gfCNCPoint6[1225] = {X 338.7767, Y 49.3353, Z -8.0000, A 0.000, B 0.000, C 0.000 }
gfCNCPoint6[1226] = {X 336.8016, Y 48.5824, Z -8.0000, A 0.000, B 0.000, C 0.000 }
gfCNCPoint6[1227] = {X 334.8992, Y 47.6612, Z -8.0000, A 0.000, B 0.000, C 0.000 }
gfCNCPoint6[1228] = {X 333.3419, Y 46.7043, Z -8.0000, A 0.000, B 0.000, C 0.000 }
gfCNCPoint6[1229] = {X 331.8606, Y 45.6336, Z -8.0000, A 0.000, B 0.000, C 0.000 }
gfCNCPoint6[1230] = {X 330.4636, Y 44.4550, Z -8.0000, A 0.000, B 0.000, C 0.000 }
gfCNCPoint6[1231] = {X 329.4664, Y 44.4078, Z -8.0000, A 0.000, B 0.000, C 0.000 }
gfCNCPoint6[1232] = {X 328.4996, Y 44.1587, Z -8.0000, A 0.000, B 0.000, C 0.000 }
gfCNCPoint6[1233] = {X 327.6038, Y 43.7181, Z -8.0000, A 0.000, B 0.000, C 0.000 }
gfCNCPoint6[1234] = {X 326.8164, Y 43.1044, Z -8.0000, A 0.000, B 0.000, C 0.000 }
gfCNCPoint6[1235] = {X 326.1897, Y 42.4934, Z -8.0000, A 0.000, B 0.000, C 0.000 }
gfCNCPoint6[1236] = {X 325.5686, Y 41.7541, Z -8.0000, A 0.000, B 0.000, C 0.000 }
gfCNCPoint6[1237] = {X 325.1052, Y 40.9070, Z -8.0000, A 0.000, B 0.000, C 0.000 }
gfCNCPoint6[1238] = {X 324.8177, Y 39.9852, Z -8.0000, A 0.000, B 0.000, C 0.000 }
gfCNCPoint6[1239] = {X 324.7172, Y 39.0249, Z -8.0000, A 0.000, B 0.000, C 0.000 }
gfCNCPoint6[1240] = {X 324.8079, Y 38.0635, Z -8.0000, A 0.000, B 0.000, C 0.000 }
gfCNCPoint6[1241] = {X 325.0860, Y 37.1389, Z -8.0000, A 0.000, B 0.000, C 0.000 }
gfCNCPoint6[1242] = {X 325.5408, Y 36.2871, Z -8.0000, A 0.000, B 0.000, C 0.000 }
gfCNCPoint6[1243] = {X 329.7765, Y 29.9537, Z -8.0000, A 0.000, B 0.000, C 0.000 }
gfCNCPoint6[1244] = {X 330.4614, Y 29.1399, Z -8.0000, A 0.000, B 0.000, C 0.000 }
gfCNCPoint6[1245] = {X 331.3063, Y 28.4938, Z -8.0000, A 0.000, B 0.000, C 0.000 }
gfCNCPoint6[1246] = {X 332.2712, Y 28.0462, Z -8.0000, A 0.000, B 0.000, C 0.000 }
gfCNCPoint6[1247] = {X 333.3101, Y 27.8182, Z -8.0000, A 0.000, B 0.000, C 0.000 }
gfCNCPoint6[1248] = {X 334.3737, Y 27.8207, Z -8.0000, A 0.000, B 0.000, C 0.000 }
gfCNCPoint6[1249] = {X 335.4115, Y 28.0536, Z -8.0000, A 0.000, B 0.000, C 0.000 }
gfCNCPoint6[1250] = {X 336.3742, Y 28.5058, Z -8.0000, A 0.000, B 0.000, C 0.000 }
gfCNCPoint6[1251] = {X 337.2161, Y 29.1558, Z -8.0000, A 0.000, B 0.000, C 0.000 }
gfCNCPoint6[1252] = {X 337.8208, Y 29.7387, Z -8.0000, A 0.000, B 0.000, C 0.000 }
gfCNCPoint6[1253] = {X 338.4966, Y 30.5667, Z -8.0000, A 0.000, B 0.000, C 0.000 }
gfCNCPoint6[1254] = {X 338.9759, Y 31.5219, Z -8.0000, A 0.000, B 0.000, C 0.000 }
gfCNCPoint6[1255] = {X 339.2358, Y 32.5585, Z -8.0000, A 0.000, B 0.000, C 0.000 }
gfCNCPoint6[1256] = {X 339.2638, Y 33.6268, Z -8.0000, A 0.000, B 0.000, C 0.000 }
gfCNCPoint6[1257] = {X 339.8716, Y 34.1825, Z -8.0000, A 0.000, B 0.000, C 0.000 }
gfCNCPoint6[1258] = {X 340.9509, Y 35.0427, Z -8.0000, A 0.000, B 0.000, C 0.000 }
gfCNCPoint6[1259] = {X 342.1372, Y 35.7481, Z -8.0000, A 0.000, B 0.000, C 0.000 }
gfCNCPoint6[1260] = {X 343.4085, Y 36.2856, Z -8.0000, A 0.000, B 0.000, C 0.000 }
gfCNCPoint6[1261] = {X 344.7410, Y 36.6452, Z -8.0000, A 0.000, B 0.000, C 0.000 }
gfCNCPoint6[1262] = {X 346.1100, Y 36.8203, Z -8.0000, A 0.000, B 0.000, C 0.000 }
gfCNCPoint6[1263] = {X 347.4901, Y 36.8075, Z -8.0000, A 0.000, B 0.000, C 0.000 }
gfCNCPoint6[1264] = {X 348.8397, Y 36.6262, Z -8.0000, A 0.000, B 0.000, C 0.000 }
gfCNCPoint6[1265] = {X 350.1418, Y 36.2276, Z -8.0000, A 0.000, B 0.000, C 0.000 }
gfCNCPoint6[1266] = {X 351.3616, Y 35.6223, Z -8.0000, A 0.000, B 0.000, C 0.000 }
gfCNCPoint6[1267] = {X 352.4665, Y 34.8263, Z -8.0000, A 0.000, B 0.000, C 0.000 }
gfCNCPoint6[1268] = {X 353.5670, Y 33.7568, Z -8.0000, A 0.000, B 0.000, C 0.000 }
gfCNCPoint6[1269] = {X 354.5194, Y 32.5535, Z -8.0000, A 0.000, B 0.000, C 0.000 }
gfCNCPoint6[1270] = {X 355.3077, Y 31.2368, Z -8.0000, A 0.000, B 0.000, C 0.000 }
gfCNCPoint6[1271] = {X 355.9184, Y 29.8290, Z -8.0000, A 0.000, B 0.000, C 0.000 }
gfCNCPoint6[1272] = {X 356.3412, Y 28.3538, Z -8.0000, A 0.000, B 0.000, C 0.000 }
gfCNCPoint6[1273] = {X 356.6058, Y 26.7186, Z -8.0000, A 0.000, B 0.000, C 0.000 }
gfCNCPoint6[1274] = {X 356.7135, Y 25.0657, Z -8.0000, A 0.000, B 0.000, C 0.000 }
gfCNCPoint6[1275] = {X 356.6634, Y 23.4100, Z -8.0000, A 0.000, B 0.000, C 0.000 }
gfCNCPoint6[1276] = {X 356.4559, Y 21.7666, Z -8.0000, A 0.000, B 0.000, C 0.000 }
gfCNCPoint6[1277] = {X 356.1193, Y 20.3212, Z -8.0000, A 0.000, B 0.000, C 0.000 }
gfCNCPoint6[1278] = {X 355.5958, Y 18.9324, Z -8.0000, A 0.000, B 0.000, C 0.000 }
gfCNCPoint6[1279] = {X 354.8945, Y 17.6245, Z -8.0000, A 0.000, B 0.000, C 0.000 }
gfCNCPoint6[1280] = {X 354.0274, Y 16.4200, Z -8.0000, A 0.000, B 0.000, C 0.000 }
gfCNCPoint6[1281] = {X 353.2099, Y 15.5491, Z -8.0000, A 0.000, B 0.000, C 0.000 }
gfCNCPoint6[1282] = {X 352.2795, Y 14.8000, Z -8.0000, A 0.000, B 0.000, C 0.000 }
gfCNCPoint6[1283] = {X 351.2542, Y 14.1872, Z -8.0000, A 0.000, B 0.000, C 0.000 }
gfCNCPoint6[1284] = {X 350.1538, Y 13.7227, Z -8.0000, A 0.000, B 0.000, C 0.000 }
gfCNCPoint6[1285] = {X 348.9996, Y 13.4152, Z -8.0000, A 0.000, B 0.000, C 0.000 }
gfCNCPoint6[1286] = {X 347.3622, Y 13.2074, Z -8.0000, A 0.000, B 0.000, C 0.000 }
gfCNCPoint6[1287] = {X 345.7117, Y 13.2121, Z -8.0000, A 0.000, B 0.000, C 0.000 }
gfCNCPoint6[1288] = {X 344.0755, Y 13.4290, Z -8.0000, A 0.000, B 0.000, C 0.000 }
gfCNCPoint6[1289] = {X 342.4808, Y 13.8547, Z -8.0000, A 0.000, B 0.000, C 0.000 }
gfCNCPoint6[1290] = {X 340.9542, Y 14.4820, Z -8.0000, A 0.000, B 0.000, C 0.000 }
gfCNCPoint6[1291] = {X 339.5209, Y 15.3006, Z -8.0000, A 0.000, B 0.000, C 0.000 }
gfCNCPoint6[1292] = {X 339.4270, Y 16.1861, Z -8.0000, A 0.000, B 0.000, C 0.000 }
gfCNCPoint6[1293] = {X 339.1738, Y 17.0397, Z -8.0000, A 0.000, B 0.000, C 0.000 }
gfCNCPoint6[1294] = {X 338.7696, Y 17.8332, Z -8.0000, A 0.000, B 0.000, C 0.000 }
gfCNCPoint6[1295] = {X 338.2280, Y 18.5400, Z -8.0000, A 0.000, B 0.000, C 0.000 }
gfCNCPoint6[1296] = {X 337.5670, Y 19.1366, Z -8.0000, A 0.000, B 0.000, C 0.000 }
gfCNCPoint6[1297] = {X 336.8400, Y 19.6716, Z -8.0000, A 0.000, B 0.000, C 0.000 }
gfCNCPoint6[1298] = {X 335.9171, Y 20.1909, Z -8.0000, A 0.000, B 0.000, C 0.000 }
gfCNCPoint6[1299] = {X 334.9039, Y 20.4988, Z -8.0000, A 0.000, B 0.000, C 0.000 }
gfCNCPoint6[1300] = {X 333.8481, Y 20.5809, Z -8.0000, A 0.000, B 0.000, C 0.000 }
gfCNCPoint6[1301] = {X 332.7995, Y 20.4334, Z -8.0000, A 0.000, B 0.000, C 0.000 }
gfCNCPoint6[1302] = {X 331.8074, Y 20.0631, Z -8.0000, A 0.000, B 0.000, C 0.000 }
gfCNCPoint6[1303] = {X 330.9186, Y 19.4876, Z -8.0000, A 0.000, B 0.000, C 0.000 }
gfCNCPoint6[1304] = {X 330.1748, Y 18.7338, Z -8.0000, A 0.000, B 0.000, C 0.000 }
gfCNCPoint6[1305] = {X 329.6111, Y 17.8373, Z -8.0000, A 0.000, B 0.000, C 0.000 }
gfCNCPoint6[1306] = {X 326.0906, Y 10.5950, Z -8.0000, A 0.000, B 0.000, C 0.000 }
gfCNCPoint6[1307] = {X 325.7555, Y 9.6856, Z -8.0000, A 0.000, B 0.000, C 0.000 }
gfCNCPoint6[1308] = {X 325.6067, Y 8.7279, Z -8.0000, A 0.000, B 0.000, C 0.000 }
gfCNCPoint6[1309] = {X 325.6502, Y 7.7596, Z -8.0000, A 0.000, B 0.000, C 0.000 }
gfCNCPoint6[1310] = {X 325.8842, Y 6.8191, Z -8.0000, A 0.000, B 0.000, C 0.000 }
gfCNCPoint6[1311] = {X 326.2994, Y 5.9433, Z -8.0000, A 0.000, B 0.000, C 0.000 }
gfCNCPoint6[1312] = {X 326.9295, Y 5.1131, Z -8.0000, A 0.000, B 0.000, C 0.000 }
gfCNCPoint6[1313] = {X 327.7216, Y 4.4356, Z -8.0000, A 0.000, B 0.000, C 0.000 }
gfCNCPoint6[1314] = {X 328.3968, Y 3.9733, Z -8.0000, A 0.000, B 0.000, C 0.000 }
gfCNCPoint6[1315] = {X 329.3289, Y 3.4830, Z -8.0000, A 0.000, B 0.000, C 0.000 }
gfCNCPoint6[1316] = {X 330.3446, Y 3.2042, Z -8.0000, A 0.000, B 0.000, C 0.000 }
gfCNCPoint6[1317] = {X 331.3964, Y 3.1497, Z -8.0000, A 0.000, B 0.000, C 0.000 }
gfCNCPoint6[1318] = {X 332.4354, Y 3.3223, Z -8.0000, A 0.000, B 0.000, C 0.000 }
gfCNCPoint6[1319] = {X 333.3715, Y 2.7957, Z -8.0000, A 0.000, B 0.000, C 0.000 }
gfCNCPoint6[1320] = {X 334.3268, Y 2.3048, Z -8.0000, A 0.000, B 0.000, C 0.000 }
gfCNCPoint6[1321] = {X 334.5381, Y 2.7358, Z -8.0000, A 0.000, B 0.000, C 0.000 }
gfCNCPoint6[1322] = {X 335.0034, Y 2.5130, Z -8.0000, A 0.000, B 0.000, C 0.000 }
gfCNCPoint6[1323] = {X 335.4728, Y 2.2988, Z -8.0000, A 0.000, B 0.000, C 0.000 }
gfCNCPoint6[1324] = {X 335.8480, Y 2.1318, Z -8.0000, A 0.000, B 0.000, C 0.000 }
gfCNCPoint6[1325] = {X 337.9512, Y 1.3113, Z -8.0000, A 0.000, B 0.000, C 0.000 }
gfCNCPoint6[1326] = {X 340.1169, Y 0.6737, Z -8.0000, A 0.000, B 0.000, C 0.000 }
gfCNCPoint6[1327] = {X 342.3292, Y 0.2238, Z -8.0000, A 0.000, B 0.000, C 0.000 }
gfCNCPoint6[1328] = {X 344.5719, Y -0.0351, Z -8.0000, A 0.000, B 0.000, C 0.000 }
gfCNCPoint6[1329] = {X 346.8285, Y -0.1013, Z -8.0000, A 0.000, B 0.000, C 0.000 }
gfCNCPoint6[1330] = {X 349.0825, Y 0.0259, Z -8.0000, A 0.000, B 0.000, C 0.000 }
gfCNCPoint6[1331] = {X 351.3173, Y 0.3455, Z -8.0000, A 0.000, B 0.000, C 0.000 }
gfCNCPoint6[1332] = {X 351.8894, Y 0.4533, Z -8.0000, A 0.000, B 0.000, C 0.000 }
gfCNCPoint6[1333] = {X 354.0191, Y 0.9988, Z -8.0000, A 0.000, B 0.000, C 0.000 }
gfCNCPoint6[1334] = {X 356.0806, Y 1.7630, Z -8.0000, A 0.000, B 0.000, C 0.000 }
gfCNCPoint6[1335] = {X 358.0513, Y 2.7375, Z -8.0000, A 0.000, B 0.000, C 0.000 }
gfCNCPoint6[1336] = {X 359.9100, Y 3.9117, Z -8.0000, A 0.000, B 0.000, C 0.000 }
gfCNCPoint6[1337] = {X 361.6364, Y 5.2730, Z -8.0000, A 0.000, B 0.000, C 0.000 }
gfCNCPoint6[1338] = {X 363.2118, Y 6.8065, Z -8.0000, A 0.000, B 0.000, C 0.000 }
gfCNCPoint6[1339] = {X 364.7640, Y 8.6820, Z -8.0000, A 0.000, B 0.000, C 0.000 }
gfCNCPoint6[1340] = {X 366.1253, Y 10.7002, Z -8.0000, A 0.000, B 0.000, C 0.000 }
gfCNCPoint6[1341] = {X 367.2828, Y 12.8419, Z -8.0000, A 0.000, B 0.000, C 0.000 }
gfCNCPoint6[1342] = {X 368.2254, Y 15.0864, Z -8.0000, A 0.000, B 0.000, C 0.000 }
gfCNCPoint6[1343] = {X 368.9440, Y 17.4124, Z -8.0000, A 0.000, B 0.000, C 0.000 }
gfCNCPoint6[1344] = {X 369.4273, Y 19.7106, Z -8.0000, A 0.000, B 0.000, C 0.000 }
gfCNCPoint6[1345] = {X 369.7390, Y 22.0383, Z -8.0000, A 0.000, B 0.000, C 0.000 }
gfCNCPoint6[1346] = {X 369.8772, Y 24.3826, Z -8.0000, A 0.000, B 0.000, C 0.000 }
gfCNCPoint6[1347] = {X 369.8413, Y 26.7308, Z -8.0000, A 0.000, B 0.000, C 0.000 }
gfCNCPoint6[1348] = {X 369.6314, Y 29.0699, Z -8.0000, A 0.000, B 0.000, C 0.000 }
gfCNCPoint6[1349] = {X 369.2488, Y 31.3870, Z -8.0000, A 0.000, B 0.000, C 0.000 }
gfCNCPoint6[1350] = {X 368.7229, Y 33.4980, Z -8.0000, A 0.000, B 0.000, C 0.000 }
gfCNCPoint6[1351] = {X 368.0128, Y 35.5544, Z -8.0000, A 0.000, B 0.000, C 0.000 }
gfCNCPoint6[1352] = {X 367.1239, Y 37.5400, Z -8.0000, A 0.000, B 0.000, C 0.000 }
gfCNCPoint6[1353] = {X 366.0631, Y 39.4394, Z -8.0000, A 0.000, B 0.000, C 0.000 }
gfCNCPoint6[1354] = {X 364.8388, Y 41.2378, Z -8.0000, A 0.000, B 0.000, C 0.000 }
gfCNCPoint6[1355] = {X 364.7204, Y 41.3994, Z -8.0000, A 0.000, B 0.000, C 0.000 }
gfCNCPoint6[1356] = {X 363.4201, Y 42.9682, Z -8.0000, A 0.000, B 0.000, C 0.000 }
gfCNCPoint6[1357] = {X 361.9805, Y 44.4103, Z -8.0000, A 0.000, B 0.000, C 0.000 }
gfCNCPoint6[1358] = {X 360.4141, Y 45.7135, Z -8.0000, A 0.000, B 0.000, C 0.000 }
gfCNCPoint6[1359] = {X 358.7341, Y 46.8667, Z -8.0000, A 0.000, B 0.000, C 0.000 }
gfCNCPoint6[1360] = {X 356.9549, Y 47.8599, Z -8.0000, A 0.000, B 0.000, C 0.000 }
gfCNCPoint6[1361] = {X 356.2499, Y 48.1934, Z -8.0000, A 0.000, B 0.000, C 0.000 }
gfCNCPoint6[1362] = {X 354.0456, Y 49.0158, Z -8.0000, A 0.000, B 0.000, C 0.000 }
gfCNCPoint6[1363] = {X 351.7691, Y 49.6098, Z -8.0000, A 0.000, B 0.000, C 0.000 }
gfCNCPoint6[1364] = {X 349.4439, Y 49.9692, Z -8.0000, A 0.000, B 0.000, C 0.000 }
gfCNCPoint6[1365] = {X 347.0943, Y 50.0903, Z -8.0000, A 0.000, B 0.000, C 0.000 }
gfCNCPoint6[1366] = {X 345.0202, Y 50.0551, Z -8.0000, A 0.000, B 0.000, C 0.000 }
gfCNCPoint6[1367] = {X 342.9569, Y 49.8401, Z -8.0000, A 0.000, B 0.000, C 0.000 }
gfCNCPoint6[1368] = {X 340.9201, Y 49.4470, Z -8.0000, A 0.000, B 0.000, C 0.000 }
gfCNCPoint6[1369] = {X 338.9250, Y 48.8787, Z -8.0000, A 0.000, B 0.000, C 0.000 }
gfCNCPoint6[1370] = {X 336.9867, Y 48.1394, Z -8.0000, A 0.000, B 0.000, C 0.000 }
gfCNCPoint6[1371] = {X 335.1199, Y 47.2348, Z -8.0000, A 0.000, B 0.000, C 0.000 }
gfCNCPoint6[1372] = {X 333.5416, Y 46.2605, Z -8.0000, A 0.000, B 0.000, C 0.000 }
gfCNCPoint6[1373] = {X 332.0435, Y 45.1668, Z -8.0000, A 0.000, B 0.000, C 0.000 }
gfCNCPoint6[1374] = {X 330.6346, Y 43.9603, Z -8.0000, A 0.000, B 0.000, C 0.000 }
gfCNCPoint6[1375] = {X 329.6760, Y 43.9518, Z -8.0000, A 0.000, B 0.000, C 0.000 }
gfCNCPoint6[1376] = {X 328.7421, Y 43.7359, Z -8.0000, A 0.000, B 0.000, C 0.000 }
gfCNCPoint6[1377] = {X 327.8770, Y 43.3228, Z -8.0000, A 0.000, B 0.000, C 0.000 }
gfCNCPoint6[1378] = {X 327.1220, Y 42.7322, Z -8.0000, A 0.000, B 0.000, C 0.000 }
gfCNCPoint6[1379] = {X 326.5249, Y 42.1498, Z -8.0000, A 0.000, B 0.000, C 0.000 }
gfCNCPoint6[1380] = {X 325.8848, Y 41.3619, Z -8.0000, A 0.000, B 0.000, C 0.000 }
gfCNCPoint6[1381] = {X 325.4424, Y 40.4483, Z -8.0000, A 0.000, B 0.000, C 0.000 }
gfCNCPoint6[1382] = {X 325.2210, Y 39.4576, Z -8.0000, A 0.000, B 0.000, C 0.000 }
gfCNCPoint6[1383] = {X 325.2326, Y 38.4426, Z -8.0000, A 0.000, B 0.000, C 0.000 }
gfCNCPoint6[1384] = {X 325.4765, Y 37.4572, Z -8.0000, A 0.000, B 0.000, C 0.000 }
gfCNCPoint6[1385] = {X 325.9397, Y 36.5539, Z -8.0000, A 0.000, B 0.000, C 0.000 }
gfCNCPoint6[1386] = {X 330.1988, Y 30.1861, Z -8.0000, A 0.000, B 0.000, C 0.000 }
gfCNCPoint6[1387] = {X 330.8195, Y 29.4619, Z -8.0000, A 0.000, B 0.000, C 0.000 }
gfCNCPoint6[1388] = {X 331.5816, Y 28.8884, Z -8.0000, A 0.000, B 0.000, C 0.000 }
gfCNCPoint6[1389] = {X 332.4494, Y 28.4927, Z -8.0000, A 0.000, B 0.000, C 0.000 }
gfCNCPoint6[1390] = {X 333.3822, Y 28.2932, Z -8.0000, A 0.000, B 0.000, C 0.000 }
gfCNCPoint6[1391] = {X 334.3359, Y 28.2995, Z -8.0000, A 0.000, B 0.000, C 0.000 }
gfCNCPoint6[1392] = {X 335.2659, Y 28.5111, Z -8.0000, A 0.000, B 0.000, C 0.000 }
gfCNCPoint6[1393] = {X 336.1285, Y 28.9182, Z -8.0000, A 0.000, B 0.000, C 0.000 }
gfCNCPoint6[1394] = {X 336.8831, Y 29.5015, Z -8.0000, A 0.000, B 0.000, C 0.000 }
gfCNCPoint6[1395] = {X 337.4845, Y 30.0811, Z -8.0000, A 0.000, B 0.000, C 0.000 }
gfCNCPoint6[1396] = {X 338.1249, Y 30.8764, Z -8.0000, A 0.000, B 0.000, C 0.000 }
gfCNCPoint6[1397] = {X 338.5647, Y 31.7978, Z -8.0000, A 0.000, B 0.000, C 0.000 }
gfCNCPoint6[1398] = {X 338.7803, Y 32.7959, Z -8.0000, A 0.000, B 0.000, C 0.000 }
gfCNCPoint6[1399] = {X 338.7601, Y 33.8167, Z -8.0000, A 0.000, B 0.000, C 0.000 }
gfCNCPoint6[1400] = {X 339.5477, Y 34.5368, Z -8.0000, A 0.000, B 0.000, C 0.000 }
gfCNCPoint6[1401] = {X 340.6406, Y 35.4108, Z -8.0000, A 0.000, B 0.000, C 0.000 }
gfCNCPoint6[1402] = {X 341.8390, Y 36.1333, Z -8.0000, A 0.000, B 0.000, C 0.000 }
gfCNCPoint6[1403] = {X 343.1221, Y 36.6917, Z -8.0000, A 0.000, B 0.000, C 0.000 }
gfCNCPoint6[1404] = {X 344.4675, Y 37.0763, Z -8.0000, A 0.000, B 0.000, C 0.000 }
gfCNCPoint6[1405] = {X 345.8519, Y 37.2804, Z -8.0000, A 0.000, B 0.000, C 0.000 }
gfCNCPoint6[1406] = {X 347.2511, Y 37.3005, Z -8.0000, A 0.000, B 0.000, C 0.000 }
gfCNCPoint6[1407] = {X 347.5149, Y 37.2868, Z -8.0000, A 0.000, B 0.000, C 0.000 }
gfCNCPoint6[1408] = {X 348.9423, Y 37.0952, Z -8.0000, A 0.000, B 0.000, C 0.000 }
gfCNCPoint6[1409] = {X 350.3194, Y 36.6736, Z -8.0000, A 0.000, B 0.000, C 0.000 }
gfCNCPoint6[1410] = {X 351.6094, Y 36.0334, Z -8.0000, A 0.000, B 0.000, C 0.000 }
gfCNCPoint6[1411] = {X 352.7779, Y 35.1916, Z -8.0000, A 0.000, B 0.000, C 0.000 }
gfCNCPoint6[1412] = {X 353.9234, Y 34.0783, Z -8.0000, A 0.000, B 0.000, C 0.000 }
gfCNCPoint6[1413] = {X 354.9147, Y 32.8258, Z -8.0000, A 0.000, B 0.000, C 0.000 }
gfCNCPoint6[1414] = {X 355.7351, Y 31.4553, Z -8.0000, A 0.000, B 0.000, C 0.000 }
gfCNCPoint6[1415] = {X 356.3706, Y 29.9899, Z -8.0000, A 0.000, B 0.000, C 0.000 }
gfCNCPoint6[1416] = {X 356.8106, Y 28.4543, Z -8.0000, A 0.000, B 0.000, C 0.000 }
gfCNCPoint6[1417] = {X 357.0827, Y 26.7727, Z -8.0000, A 0.000, B 0.000, C 0.000 }
gfCNCPoint6[1418] = {X 357.1934, Y 25.0729, Z -8.0000, A 0.000, B 0.000, C 0.000 }
gfCNCPoint6[1419] = {X 357.1417, Y 23.3702, Z -8.0000, A 0.000, B 0.000, C 0.000 }
gfCNCPoint6[1420] = {X 356.9281, Y 21.6801, Z -8.0000, A 0.000, B 0.000, C 0.000 }
gfCNCPoint6[1421] = {X 356.5766, Y 20.1750, Z -8.0000, A 0.000, B 0.000, C 0.000 }
gfCNCPoint6[1422] = {X 356.0306, Y 18.7290, Z -8.0000, A 0.000, B 0.000, C 0.000 }
gfCNCPoint6[1423] = {X 355.2997, Y 17.3672, Z -8.0000, A 0.000, B 0.000, C 0.000 }
gfCNCPoint6[1424] = {X 354.3964, Y 16.1130, Z -8.0000, A 0.000, B 0.000, C 0.000 }
gfCNCPoint6[1425] = {X 353.5334, Y 15.1945, Z -8.0000, A 0.000, B 0.000, C 0.000 }
gfCNCPoint6[1426] = {X 352.5515, Y 14.4045, Z -8.0000, A 0.000, B 0.000, C 0.000 }
gfCNCPoint6[1427] = {X 351.4695, Y 13.7582, Z -8.0000, A 0.000, B 0.000, C 0.000 }
gfCNCPoint6[1428] = {X 350.3084, Y 13.2682, Z -8.0000, A 0.000, B 0.000, C 0.000 }
gfCNCPoint6[1429] = {X 349.0905, Y 12.9439, Z -8.0000, A 0.000, B 0.000, C 0.000 }
gfCNCPoint6[1430] = {X 347.3478, Y 12.7257, Z -8.0000, A 0.000, B 0.000, C 0.000 }
gfCNCPoint6[1431] = {X 345.5916, Y 12.7394, Z -8.0000, A 0.000, B 0.000, C 0.000 }
gfCNCPoint6[1432] = {X 343.8525, Y 12.9846, Z -8.0000, A 0.000, B 0.000, C 0.000 }
gfCNCPoint6[1433] = {X 342.1610, Y 13.4573, Z -8.0000, A 0.000, B 0.000, C 0.000 }
gfCNCPoint6[1434] = {X 340.5466, Y 14.1489, Z -8.0000, A 0.000, B 0.000, C 0.000 }
gfCNCPoint6[1435] = {X 339.0376, Y 15.0476, Z -8.0000, A 0.000, B 0.000, C 0.000 }
gfCNCPoint6[1436] = {X 338.9894, Y 15.9053, Z -8.0000, A 0.000, B 0.000, C 0.000 }
gfCNCPoint6[1437] = {X 338.7755, Y 16.7372, Z -8.0000, A 0.000, B 0.000, C 0.000 }
gfCNCPoint6[1438] = {X 338.4040, Y 17.5118, Z -8.0000, A 0.000, B 0.000, C 0.000 }
gfCNCPoint6[1439] = {X 337.8891, Y 18.1994, Z -8.0000, A 0.000, B 0.000, C 0.000 }
gfCNCPoint6[1440] = {X 337.2504, Y 18.7738, Z -8.0000, A 0.000, B 0.000, C 0.000 }
gfCNCPoint6[1441] = {X 336.5606, Y 19.2813, Z -8.0000, A 0.000, B 0.000, C 0.000 }
gfCNCPoint6[1442] = {X 335.7284, Y 19.7495, Z -8.0000, A 0.000, B 0.000, C 0.000 }
gfCNCPoint6[1443] = {X 334.8148, Y 20.0271, Z -8.0000, A 0.000, B 0.000, C 0.000 }
gfCNCPoint6[1444] = {X 333.8628, Y 20.1012, Z -8.0000, A 0.000, B 0.000, C 0.000 }
gfCNCPoint6[1445] = {X 332.9173, Y 19.9681, Z -8.0000, A 0.000, B 0.000, C 0.000 }
gfCNCPoint6[1446] = {X 332.0228, Y 19.6341, Z -8.0000, A 0.000, B 0.000, C 0.000 }
gfCNCPoint6[1447] = {X 331.2213, Y 19.1151, Z -8.0000, A 0.000, B 0.000, C 0.000 }
gfCNCPoint6[1448] = {X 330.5507, Y 18.4353, Z -8.0000, A 0.000, B 0.000, C 0.000 }
gfCNCPoint6[1449] = {X 330.0425, Y 17.6269, Z -8.0000, A 0.000, B 0.000, C 0.000 }
gfCNCPoint6[1450] = {X 326.5223, Y 10.3852, Z -8.0000, A 0.000, B 0.000, C 0.000 }
gfCNCPoint6[1451] = {X 326.2154, Y 9.5469, Z -8.0000, A 0.000, B 0.000, C 0.000 }
gfCNCPoint6[1452] = {X 326.0841, Y 8.6639, Z -8.0000, A 0.000, B 0.000, C 0.000 }
gfCNCPoint6[1453] = {X 326.1338, Y 7.7725, Z -8.0000, A 0.000, B 0.000, C 0.000 }
gfCNCPoint6[1454] = {X 326.3623, Y 6.9096, Z -8.0000, A 0.000, B 0.000, C 0.000 }
gfCNCPoint6[1455] = {X 326.7603, Y 6.1105, Z -8.0000, A 0.000, B 0.000, C 0.000 }
gfCNCPoint6[1456] = {X 327.3114, Y 5.4082, Z -8.0000, A 0.000, B 0.000, C 0.000 }
gfCNCPoint6[1457] = {X 327.9929, Y 4.8316, Z -8.0000, A 0.000, B 0.000, C 0.000 }
gfCNCPoint6[1458] = {X 328.6647, Y 4.3715, Z -8.0000, A 0.000, B 0.000, C 0.000 }
gfCNCPoint6[1459] = {X 329.5520, Y 3.9113, Z -8.0000, A 0.000, B 0.000, C 0.000 }
gfCNCPoint6[1460] = {X 330.5202, Y 3.6632, Z -8.0000, A 0.000, B 0.000, C 0.000 }
gfCNCPoint6[1461] = {X 331.5195, Y 3.6400, Z -8.0000, A 0.000, B 0.000, C 0.000 }
gfCNCPoint6[1462] = {X 332.4982, Y 3.8430, Z -8.0000, A 0.000, B 0.000, C 0.000 }
gfCNCPoint6[1463] = {X 333.5066, Y 3.2683, Z -8.0000, A 0.000, B 0.000, C 0.000 }
gfCNCPoint6[1464] = {X 334.5381, Y 2.7358, Z -8.0000, A 0.000, B 0.000, C 0.000 }
gfCNCPoint6[1465] = {X 334.3268, Y 2.3048, Z -8.0000, A 0.000, B 0.000, C 0.000 }
gfCNCPoint6[1466] = {X 2.3033, Y 2.3048, Z -8.0000, A 0.000, B 0.000, C 0.000 }
gfCNCPoint6[1467] = {X 2.3033, Y 6.8597, Z -8.0000, A 0.000, B 0.000, C 0.000 }
gfCNCPoint6[1468] = {X 2.4157, Y 6.8822, Z -8.0000, A 0.000, B 0.000, C 0.000 }
gfCNCPoint6[1469] = {X 4.7212, Y 6.0042, Z -8.0000, A 0.000, B 0.000, C 0.000 }
gfCNCPoint6[1470] = {X 7.0988, Y 5.3462, Z -8.0000, A 0.000, B 0.000, C 0.000 }
gfCNCPoint6[1471] = {X 9.5276, Y 4.9141, Z -8.0000, A 0.000, B 0.000, C 0.000 }
gfCNCPoint6[1472] = {X 11.9863, Y 4.7116, Z -8.0000, A 0.000, B 0.000, C 0.000 }
gfCNCPoint6[1473] = {X 14.4531, Y 4.7406, Z -8.0000, A 0.000, B 0.000, C 0.000 }
gfCNCPoint6[1474] = {X 16.9064, Y 5.0008, Z -8.0000, A 0.000, B 0.000, C 0.000 }
gfCNCPoint6[1475] = {X 18.9221, Y 5.4146, Z -8.0000, A 0.000, B 0.000, C 0.000 }
gfCNCPoint6[1476] = {X 20.8843, Y 6.0345, Z -8.0000, A 0.000, B 0.000, C 0.000 }
gfCNCPoint6[1477] = {X 22.7719, Y 6.8540, Z -8.0000, A 0.000, B 0.000, C 0.000 }
gfCNCPoint6[1478] = {X 24.4916, Y 7.8179, Z -8.0000, A 0.000, B 0.000, C 0.000 }
gfCNCPoint6[1479] = {X 26.1074, Y 8.9475, Z -8.0000, A 0.000, B 0.000, C 0.000 }
gfCNCPoint6[1480] = {X 27.4014, Y 10.0778, Z -8.0000, A 0.000, B 0.000, C 0.000 }
gfCNCPoint6[1481] = {X 28.5623, Y 11.3446, Z -8.0000, A 0.000, B 0.000, C 0.000 }
gfCNCPoint6[1482] = {X 29.5756, Y 12.7322, Z -8.0000, A 0.000, B 0.000, C 0.000 }
gfCNCPoint6[1483] = {X 30.4290, Y 14.2234, Z -8.0000, A 0.000, B 0.000, C 0.000 }
gfCNCPoint6[1484] = {X 31.1119, Y 15.8001, Z -8.0000, A 0.000, B 0.000, C 0.000 }
gfCNCPoint6[1485] = {X 31.6714, Y 17.7359, Z -8.0000, A 0.000, B 0.000, C 0.000 }
gfCNCPoint6[1486] = {X 32.0045, Y 19.7231, Z -8.0000, A 0.000, B 0.000, C 0.000 }
gfCNCPoint6[1487] = {X 32.1068, Y 21.7355, Z -8.0000, A 0.000, B 0.000, C 0.000 }
gfCNCPoint6[1488] = {X 31.9770, Y 23.7463, Z -8.0000, A 0.000, B 0.000, C 0.000 }
gfCNCPoint6[1489] = {X 31.6168, Y 25.7288, Z -8.0000, A 0.000, B 0.000, C 0.000 }
gfCNCPoint6[1490] = {X 31.1975, Y 27.1578, Z -8.0000, A 0.000, B 0.000, C 0.000 }
gfCNCPoint6[1491] = {X 30.6307, Y 28.5350, Z -8.0000, A 0.000, B 0.000, C 0.000 }
gfCNCPoint6[1492] = {X 29.9226, Y 29.8451, Z -8.0000, A 0.000, B 0.000, C 0.000 }
gfCNCPoint6[1493] = {X 29.0809, Y 31.0737, Z -8.0000, A 0.000, B 0.000, C 0.000 }
gfCNCPoint6[1494] = {X 29.6386, Y 31.7920, Z -8.0000, A 0.000, B 0.000, C 0.000 }
gfCNCPoint6[1495] = {X 30.0954, Y 32.5783, Z -8.0000, A 0.000, B 0.000, C 0.000 }
gfCNCPoint6[1496] = {X 33.1423, Y 38.8726, Z -8.0000, A 0.000, B 0.000, C 0.000 }
gfCNCPoint6[1497] = {X 33.5391, Y 39.8957, Z -8.0000, A 0.000, B 0.000, C 0.000 }
gfCNCPoint6[1498] = {X 33.7662, Y 40.9694, Z -8.0000, A 0.000, B 0.000, C 0.000 }
gfCNCPoint6[1499] = {X 33.8177, Y 42.0656, Z -8.0000, A 0.000, B 0.000, C 0.000 }
gfCNCPoint6[1500] = {X 33.7164, Y 43.0266, Z -8.0000, A 0.000, B 0.000, C 0.000 }
gfCNCPoint6[1501] = {X 33.4799, Y 43.9636, Z -8.0000, A 0.000, B 0.000, C 0.000 }
gfCNCPoint6[1502] = {X 33.1103, Y 44.8630, Z -8.0000, A 0.000, B 0.000, C 0.000 }
gfCNCPoint6[1503] = {X 32.6161, Y 45.7005, Z -8.0000, A 0.000, B 0.000, C 0.000 }
gfCNCPoint6[1504] = {X 32.0075, Y 46.4590, Z -8.0000, A 0.000, B 0.000, C 0.000 }
gfCNCPoint6[1505] = {X 31.2970, Y 47.1229, Z -8.0000, A 0.000, B 0.000, C 0.000 }
gfCNCPoint6[1506] = {X 30.7618, Y 47.5557, Z -8.0000, A 0.000, B 0.000, C 0.000 }
gfCNCPoint6[1507] = {X 29.8560, Y 48.1750, Z -8.0000, A 0.000, B 0.000, C 0.000 }
gfCNCPoint6[1508] = {X 28.8625, Y 48.6408, Z -8.0000, A 0.000, B 0.000, C 0.000 }
gfCNCPoint6[1509] = {X 27.8070, Y 48.9409, Z -8.0000, A 0.000, B 0.000, C 0.000 }
gfCNCPoint6[1510] = {X 26.7171, Y 49.0676, Z -8.0000, A 0.000, B 0.000, C 0.000 }
gfCNCPoint6[1511] = {X 25.6209, Y 49.0176, Z -8.0000, A 0.000, B 0.000, C 0.000 }
gfCNCPoint6[1512] = {X 23.9297, Y 49.8561, Z -8.0000, A 0.000, B 0.000, C 0.000 }
gfCNCPoint6[1513] = {X 22.1918, Y 50.5932, Z -8.0000, A 0.000, B 0.000, C 0.000 }
gfCNCPoint6[1514] = {X 20.4134, Y 51.2261, Z -8.0000, A 0.000, B 0.000, C 0.000 }
gfCNCPoint6[1515] = {X 18.2642, Y 51.8320, Z -8.0000, A 0.000, B 0.000, C 0.000 }
gfCNCPoint6[1516] = {X 16.0699, Y 52.2456, Z -8.0000, A 0.000, B 0.000, C 0.000 }
gfCNCPoint6[1517] = {X 13.8475, Y 52.4636, Z -8.0000, A 0.000, B 0.000, C 0.000 }
gfCNCPoint6[1518] = {X 11.6147, Y 52.4842, Z -8.0000, A 0.000, B 0.000, C 0.000 }
gfCNCPoint6[1519] = {X 9.3887, Y 52.3073, Z -8.0000, A 0.000, B 0.000, C 0.000 }
gfCNCPoint6[1520] = {X 7.1871, Y 51.9343, Z -8.0000, A 0.000, B 0.000, C 0.000 }
gfCNCPoint6[1521] = {X 6.2986, Y 51.7240, Z -8.0000, A 0.000, B 0.000, C 0.000 }
gfCNCPoint6[1522] = {X 5.4212, Y 51.4717, Z -8.0000, A 0.000, B 0.000, C 0.000 }
gfCNCPoint6[1523] = {X 3.8339, Y 50.8964, Z -8.0000, A 0.000, B 0.000, C 0.000 }
gfCNCPoint6[1524] = {X 2.3033, Y 50.1837, Z -8.0000, A 0.000, B 0.000, C 0.000 }
gfCNCPoint6[1525] = {X 2.3033, Y 97.6952, Z -8.0000, A 0.000, B 0.000, C 0.000 }
gfCNCPoint6[1526] = {X 120.1200, Y 97.6952, Z -8.0000, A 0.000, B 0.000, C 0.000 }
gfCNCPoint6[1527] = {X 120.1200, Y 97.0659, Z -8.0000, A 0.000, B 0.000, C 0.000 }
gfCNCPoint6[1528] = {X 120.2337, Y 96.0189, Z -8.0000, A 0.000, B 0.000, C 0.000 }
gfCNCPoint6[1529] = {X 120.5693, Y 95.0206, Z -8.0000, A 0.000, B 0.000, C 0.000 }
gfCNCPoint6[1530] = {X 121.1113, Y 94.1176, Z -8.0000, A 0.000, B 0.000, C 0.000 }
gfCNCPoint6[1531] = {X 121.8345, Y 93.3519, Z -8.0000, A 0.000, B 0.000, C 0.000 }
gfCNCPoint6[1532] = {X 122.7051, Y 92.7592, Z -8.0000, A 0.000, B 0.000, C 0.000 }
gfCNCPoint6[1533] = {X 123.6826, Y 92.3671, Z -8.0000, A 0.000, B 0.000, C 0.000 }
gfCNCPoint6[1534] = {X 124.7214, Y 92.1939, Z -8.0000, A 0.000, B 0.000, C 0.000 }
gfCNCPoint6[1535] = {X 124.7830, Y 92.1778, Z -8.0000, A 0.000, B 0.000, C 0.000 }
gfCNCPoint6[1536] = {X 124.8455, Y 92.1662, Z -8.0000, A 0.000, B 0.000, C 0.000 }
gfCNCPoint6[1537] = {X 125.3649, Y 92.0892, Z -8.0000, A 0.000, B 0.000, C 0.000 }
gfCNCPoint6[1538] = {X 126.0999, Y 91.9677, Z -8.0000, A 0.000, B 0.000, C 0.000 }
gfCNCPoint6[1539] = {X 126.8258, Y 91.8004, Z -8.0000, A 0.000, B 0.000, C 0.000 }
gfCNCPoint6[1540] = {X 127.9391, Y 90.7466, Z -8.0000, A 0.000, B 0.000, C 0.000 }
gfCNCPoint6[1541] = {X 128.9956, Y 89.6359, Z -8.0000, A 0.000, B 0.000, C 0.000 }
gfCNCPoint6[1542] = {X 154.9456, Y 61.1412, Z -8.0000, A 0.000, B 0.000, C 0.000 }
gfCNCPoint6[1543] = {X 154.6590, Y 60.4489, Z -8.0000, A 0.000, B 0.000, C 0.000 }
gfCNCPoint6[1544] = {X 154.4818, Y 59.7209, Z -8.0000, A 0.000, B 0.000, C 0.000 }
gfCNCPoint6[1545] = {X 154.4181, Y 58.9744, Z -8.0000, A 0.000, B 0.000, C 0.000 }
gfCNCPoint6[1546] = {X 154.4180, Y 58.0000, Z -8.0000, A 0.000, B 0.000, C 0.000 }
gfCNCPoint6[1547] = {X 154.5117, Y 57.0480, Z -8.0000, A 0.000, B 0.000, C 0.000 }
gfCNCPoint6[1548] = {X 154.7894, Y 56.1325, Z -8.0000, A 0.000, B 0.000, C 0.000 }
gfCNCPoint6[1549] = {X 155.2404, Y 55.2888, Z -8.0000, A 0.000, B 0.000, C 0.000 }
gfCNCPoint6[1550] = {X 155.8473, Y 54.5493, Z -8.0000, A 0.000, B 0.000, C 0.000 }
gfCNCPoint6[1551] = {X 156.5868, Y 53.9424, Z -8.0000, A 0.000, B 0.000, C 0.000 }
gfCNCPoint6[1552] = {X 157.4305, Y 53.4915, Z -8.0000, A 0.000, B 0.000, C 0.000 }
gfCNCPoint6[1553] = {X 158.3459, Y 53.2138, Z -8.0000, A 0.000, B 0.000, C 0.000 }
gfCNCPoint6[1554] = {X 159.2980, Y 53.1200, Z -8.0000, A 0.000, B 0.000, C 0.000 }
gfCNCPoint6[1555] = {X 178.5335, Y 53.1200, Z -8.0000, A 0.000, B 0.000, C 0.000 }
gfCNCPoint6[1556] = {X 179.4855, Y 53.2138, Z -8.0000, A 0.000, B 0.000, C 0.000 }
gfCNCPoint6[1557] = {X 180.4010, Y 53.4915, Z -8.0000, A 0.000, B 0.000, C 0.000 }
gfCNCPoint6[1558] = {X 181.2447, Y 53.9424, Z -8.0000, A 0.000, B 0.000, C 0.000 }
gfCNCPoint6[1559] = {X 181.9842, Y 54.5493, Z -8.0000, A 0.000, B 0.000, C 0.000 }
gfCNCPoint6[1560] = {X 182.5911, Y 55.2888, Z -8.0000, A 0.000, B 0.000, C 0.000 }
gfCNCPoint6[1561] = {X 183.0420, Y 56.1325, Z -8.0000, A 0.000, B 0.000, C 0.000 }
gfCNCPoint6[1562] = {X 183.3197, Y 57.0480, Z -8.0000, A 0.000, B 0.000, C 0.000 }
gfCNCPoint6[1563] = {X 183.4135, Y 58.0000, Z -8.0000, A 0.000, B 0.000, C 0.000 }
gfCNCPoint6[1564] = {X 183.4133, Y 58.9744, Z -8.0000, A 0.000, B 0.000, C 0.000 }
gfCNCPoint6[1565] = {X 183.3513, Y 59.7109, Z -8.0000, A 0.000, B 0.000, C 0.000 }
gfCNCPoint6[1566] = {X 183.1787, Y 60.4296, Z -8.0000, A 0.000, B 0.000, C 0.000 }
gfCNCPoint6[1567] = {X 182.8996, Y 61.1140, Z -8.0000, A 0.000, B 0.000, C 0.000 }
gfCNCPoint6[1568] = {X 209.7071, Y 90.3786, Z -8.0000, A 0.000, B 0.000, C 0.000 }
gfCNCPoint6[1569] = {X 210.3586, Y 91.0534, Z -8.0000, A 0.000, B 0.000, C 0.000 }
gfCNCPoint6[1570] = {X 211.0445, Y 91.6932, Z -8.0000, A 0.000, B 0.000, C 0.000 }
gfCNCPoint6[1571] = {X 211.3202, Y 91.8798, Z -8.0000, A 0.000, B 0.000, C 0.000 }
gfCNCPoint6[1572] = {X 211.6345, Y 91.9895, Z -8.0000, A 0.000, B 0.000, C 0.000 }
gfCNCPoint6[1573] = {X 212.1999, Y 92.1079, Z -8.0000, A 0.000, B 0.000, C 0.000 }
gfCNCPoint6[1574] = {X 213.3864, Y 92.2574, Z -8.0000, A 0.000, B 0.000, C 0.000 }
gfCNCPoint6[1575] = {X 214.4302, Y 92.1753, Z -8.0000, A 0.000, B 0.000, C 0.000 }
gfCNCPoint6[1576] = {X 215.4756, Y 92.1151, Z -8.0000, A 0.000, B 0.000, C 0.000 }
gfCNCPoint6[1577] = {X 216.0506, Y 92.0559, Z -8.0000, A 0.000, B 0.000, C 0.000 }
gfCNCPoint6[1578] = {X 216.6045, Y 91.8906, Z -8.0000, A 0.000, B 0.000, C 0.000 }
gfCNCPoint6[1579] = {X 217.1178, Y 91.6249, Z -8.0000, A 0.000, B 0.000, C 0.000 }
gfCNCPoint6[1580] = {X 244.5995, Y 74.0197, Z -8.0000, A 0.000, B 0.000, C 0.000 }
gfCNCPoint6[1581] = {X 221.4279, Y 64.9271, Z -8.0000, A 0.000, B 0.000, C 0.000 }
gfCNCPoint6[1582] = {X 219.7197, Y 64.3550, Z -8.0000, A 0.000, B 0.000, C 0.000 }
gfCNCPoint6[1583] = {X 217.9575, Y 63.9814, Z -8.0000, A 0.000, B 0.000, C 0.000 }
gfCNCPoint6[1584] = {X 216.1642, Y 63.8112, Z -8.0000, A 0.000, B 0.000, C 0.000 }
gfCNCPoint6[1585] = {X 215.1117, Y 63.6593, Z -8.0000, A 0.000, B 0.000, C 0.000 }
gfCNCPoint6[1586] = {X 214.1171, Y 63.2831, Z -8.0000, A 0.000, B 0.000, C 0.000 }
gfCNCPoint6[1587] = {X 213.2276, Y 62.7003, Z -8.0000, A 0.000, B 0.000, C 0.000 }
gfCNCPoint6[1588] = {X 212.4855, Y 61.9387, Z -8.0000, A 0.000, B 0.000, C 0.000 }
gfCNCPoint6[1589] = {X 211.9259, Y 61.0344, Z -8.0000, A 0.000, B 0.000, C 0.000 }
gfCNCPoint6[1590] = {X 211.5756, Y 60.0304, Z -8.0000, A 0.000, B 0.000, C 0.000 }
gfCNCPoint6[1591] = {X 211.4510, Y 58.9744, Z -8.0000, A 0.000, B 0.000, C 0.000 }
gfCNCPoint6[1592] = {X 211.4508, Y 58.0000, Z -8.0000, A 0.000, B 0.000, C 0.000 }
gfCNCPoint6[1593] = {X 211.5446, Y 57.0480, Z -8.0000, A 0.000, B 0.000, C 0.000 }
gfCNCPoint6[1594] = {X 211.8223, Y 56.1325, Z -8.0000, A 0.000, B 0.000, C 0.000 }
gfCNCPoint6[1595] = {X 212.2732, Y 55.2888, Z -8.0000, A 0.000, B 0.000, C 0.000 }
gfCNCPoint6[1596] = {X 212.8801, Y 54.5493, Z -8.0000, A 0.000, B 0.000, C 0.000 }
gfCNCPoint6[1597] = {X 213.6196, Y 53.9424, Z -8.0000, A 0.000, B 0.000, C 0.000 }
gfCNCPoint6[1598] = {X 214.4633, Y 53.4915, Z -8.0000, A 0.000, B 0.000, C 0.000 }
gfCNCPoint6[1599] = {X 215.3788, Y 53.2138, Z -8.0000, A 0.000, B 0.000, C 0.000 }
gfCNCPoint6[1600] = {X 216.3308, Y 53.1200, Z -8.0000, A 0.000, B 0.000, C 0.000 }
gfCNCPoint6[1601] = {X 237.2617, Y 53.1200, Z -8.0000, A 0.000, B 0.000, C 0.000 }
gfCNCPoint6[1602] = {X 238.3264, Y 53.2376, Z -8.0000, A 0.000, B 0.000, C 0.000 }
gfCNCPoint6[1603] = {X 239.3398, Y 53.5846, Z -8.0000, A 0.000, B 0.000, C 0.000 }
gfCNCPoint6[1604] = {X 240.2531, Y 54.1444, Z -8.0000, A 0.000, B 0.000, C 0.000 }
gfCNCPoint6[1605] = {X 241.0222, Y 54.8899, Z -8.0000, A 0.000, B 0.000, C 0.000 }
gfCNCPoint6[1606] = {X 241.6102, Y 55.7853, Z -8.0000, A 0.000, B 0.000, C 0.000 }
gfCNCPoint6[1607] = {X 241.9886, Y 56.7874, Z -8.0000, A 0.000, B 0.000, C 0.000 }
gfCNCPoint6[1608] = {X 242.1393, Y 57.8479, Z -8.0000, A 0.000, B 0.000, C 0.000 }
gfCNCPoint6[1609] = {X 248.3226, Y 60.2591, Z -8.0000, A 0.000, B 0.000, C 0.000 }
gfCNCPoint6[1610] = {X 275.0715, Y 70.8763, Z -8.0000, A 0.000, B 0.000, C 0.000 }
gfCNCPoint6[1611] = {X 275.0713, Y 63.6739, Z -8.0000, A 0.000, B 0.000, C 0.000 }
gfCNCPoint6[1612] = {X 274.0633, Y 63.3054, Z -8.0000, A 0.000, B 0.000, C 0.000 }
gfCNCPoint6[1613] = {X 273.1602, Y 62.7254, Z -8.0000, A 0.000, B 0.000, C 0.000 }
gfCNCPoint6[1614] = {X 272.4058, Y 61.9621, Z -8.0000, A 0.000, B 0.000, C 0.000 }
gfCNCPoint6[1615] = {X 271.8364, Y 61.0523, Z -8.0000, A 0.000, B 0.000, C 0.000 }
gfCNCPoint6[1616] = {X 271.4797, Y 60.0401, Z -8.0000, A 0.000, B 0.000, C 0.000 }
gfCNCPoint6[1617] = {X 271.3529, Y 58.9744, Z -8.0000, A 0.000, B 0.000, C 0.000 }
gfCNCPoint6[1618] = {X 271.3527, Y 58.0000, Z -8.0000, A 0.000, B 0.000, C 0.000 }
gfCNCPoint6[1619] = {X 271.4465, Y 57.0480, Z -8.0000, A 0.000, B 0.000, C 0.000 }
gfCNCPoint6[1620] = {X 271.7242, Y 56.1325, Z -8.0000, A 0.000, B 0.000, C 0.000 }
gfCNCPoint6[1621] = {X 272.1751, Y 55.2888, Z -8.0000, A 0.000, B 0.000, C 0.000 }
gfCNCPoint6[1622] = {X 272.7820, Y 54.5493, Z -8.0000, A 0.000, B 0.000, C 0.000 }
gfCNCPoint6[1623] = {X 273.5215, Y 53.9424, Z -8.0000, A 0.000, B 0.000, C 0.000 }
gfCNCPoint6[1624] = {X 274.3652, Y 53.4915, Z -8.0000, A 0.000, B 0.000, C 0.000 }
gfCNCPoint6[1625] = {X 275.2806, Y 53.2138, Z -8.0000, A 0.000, B 0.000, C 0.000 }
gfCNCPoint6[1626] = {X 276.2327, Y 53.1200, Z -8.0000, A 0.000, B 0.000, C 0.000 }
gfCNCPoint6[1627] = {X 292.7731, Y 53.1200, Z -8.0000, A 0.000, B 0.000, C 0.000 }
gfCNCPoint6[1628] = {X 293.7251, Y 53.2138, Z -8.0000, A 0.000, B 0.000, C 0.000 }
gfCNCPoint6[1629] = {X 294.6406, Y 53.4915, Z -8.0000, A 0.000, B 0.000, C 0.000 }
gfCNCPoint6[1630] = {X 295.4843, Y 53.9424, Z -8.0000, A 0.000, B 0.000, C 0.000 }
gfCNCPoint6[1631] = {X 296.2238, Y 54.5493, Z -8.0000, A 0.000, B 0.000, C 0.000 }
gfCNCPoint6[1632] = {X 296.8307, Y 55.2888, Z -8.0000, A 0.000, B 0.000, C 0.000 }
gfCNCPoint6[1633] = {X 297.2816, Y 56.1325, Z -8.0000, A 0.000, B 0.000, C 0.000 }
gfCNCPoint6[1634] = {X 297.5593, Y 57.0480, Z -8.0000, A 0.000, B 0.000, C 0.000 }
gfCNCPoint6[1635] = {X 297.6531, Y 58.0000, Z -8.0000, A 0.000, B 0.000, C 0.000 }
gfCNCPoint6[1636] = {X 297.6531, Y 58.9364, Z -8.0000, A 0.000, B 0.000, C 0.000 }
gfCNCPoint6[1637] = {X 297.5313, Y 60.0088, Z -8.0000, A 0.000, B 0.000, C 0.000 }
gfCNCPoint6[1638] = {X 297.1775, Y 61.0285, Z -8.0000, A 0.000, B 0.000, C 0.000 }
gfCNCPoint6[1639] = {X 296.6088, Y 61.9458, Z -8.0000, A 0.000, B 0.000, C 0.000 }
gfCNCPoint6[1640] = {X 295.8530, Y 62.7163, Z -8.0000, A 0.000, B 0.000, C 0.000 }
gfCNCPoint6[1641] = {X 294.9468, Y 63.3025, Z -8.0000, A 0.000, B 0.000, C 0.000 }
gfCNCPoint6[1642] = {X 293.9341, Y 63.6758, Z -8.0000, A 0.000, B 0.000, C 0.000 }
gfCNCPoint6[1643] = {X 293.9341, Y 92.3190, Z -8.0000, A 0.000, B 0.000, C 0.000 }
gfCNCPoint6[1644] = {X 294.9459, Y 92.6946, Z -8.0000, A 0.000, B 0.000, C 0.000 }
gfCNCPoint6[1645] = {X 295.8513, Y 93.2821, Z -8.0000, A 0.000, B 0.000, C 0.000 }
gfCNCPoint6[1646] = {X 296.6065, Y 94.0531, Z -8.0000, A 0.000, B 0.000, C 0.000 }
gfCNCPoint6[1647] = {X 297.1751, Y 94.9705, Z -8.0000, A 0.000, B 0.000, C 0.000 }
gfCNCPoint6[1648] = {X 297.5297, Y 95.9898, Z -8.0000, A 0.000, B 0.000, C 0.000 }
gfCNCPoint6[1649] = {X 297.6531, Y 97.0620, Z -8.0000, A 0.000, B 0.000, C 0.000 }
gfCNCPoint6[1650] = {X 297.6531, Y 97.6952, Z -8.0000, A 0.000, B 0.000, C 0.000 }
gfCNCPoint6[1651] = {X 297.1731, Y 97.6952, Z -8.0000, A 0.000, B 0.000, C 0.000 }
gfCNCPoint6[1652] = {X 297.1731, Y 98.0000, Z -8.0000, A 0.000, B 0.000, C 0.000 }
gfCNCPoint6[1653] = {X 297.0628, Y 98.9791, Z -8.0000, A 0.000, B 0.000, C 0.000 }
gfCNCPoint6[1654] = {X 296.7373, Y 99.9091, Z -8.0000, A 0.000, B 0.000, C 0.000 }
gfCNCPoint6[1655] = {X 296.2131, Y 100.7434, Z -8.0000, A 0.000, B 0.000, C 0.000 }
gfCNCPoint6[1656] = {X 295.5164, Y 101.4401, Z -8.0000, A 0.000, B 0.000, C 0.000 }
gfCNCPoint6[1657] = {X 294.6822, Y 101.9643, Z -8.0000, A 0.000, B 0.000, C 0.000 }
gfCNCPoint6[1658] = {X 293.7522, Y 102.2897, Z -8.0000, A 0.000, B 0.000, C 0.000 }
gfCNCPoint6[1659] = {X 292.7731, Y 102.4000, Z -8.0000, A 0.000, B 0.000, C 0.000 }
gfCNCPoint6[1660] = {X 276.2327, Y 102.4000, Z -8.0000, A 0.000, B 0.000, C 0.000 }
gfCNCPoint6[1661] = {X 275.2536, Y 102.2897, Z -8.0000, A 0.000, B 0.000, C 0.000 }
gfCNCPoint6[1662] = {X 274.3236, Y 101.9643, Z -8.0000, A 0.000, B 0.000, C 0.000 }
gfCNCPoint6[1663] = {X 273.4893, Y 101.4401, Z -8.0000, A 0.000, B 0.000, C 0.000 }
gfCNCPoint6[1664] = {X 272.7926, Y 100.7434, Z -8.0000, A 0.000, B 0.000, C 0.000 }
gfCNCPoint6[1665] = {X 272.2684, Y 99.9091, Z -8.0000, A 0.000, B 0.000, C 0.000 }
gfCNCPoint6[1666] = {X 271.9430, Y 98.9791, Z -8.0000, A 0.000, B 0.000, C 0.000 }
gfCNCPoint6[1667] = {X 271.8327, Y 98.0000, Z -8.0000, A 0.000, B 0.000, C 0.000 }
gfCNCPoint6[1668] = {X 271.8329, Y 97.0190, Z -8.0000, A 0.000, B 0.000, C 0.000 }
gfCNCPoint6[1669] = {X 271.9305, Y 96.1432, Z -8.0000, A 0.000, B 0.000, C 0.000 }
gfCNCPoint6[1670] = {X 272.2006, Y 95.3045, Z -8.0000, A 0.000, B 0.000, C 0.000 }
gfCNCPoint6[1671] = {X 272.6325, Y 94.5364, Z -8.0000, A 0.000, B 0.000, C 0.000 }
gfCNCPoint6[1672] = {X 273.2087, Y 93.8698, Z -8.0000, A 0.000, B 0.000, C 0.000 }
gfCNCPoint6[1673] = {X 273.9062, Y 93.3313, Z -8.0000, A 0.000, B 0.000, C 0.000 }
gfCNCPoint6[1674] = {X 274.6970, Y 92.9426, Z -8.0000, A 0.000, B 0.000, C 0.000 }
gfCNCPoint6[1675] = {X 275.5494, Y 92.7193, Z -8.0000, A 0.000, B 0.000, C 0.000 }
gfCNCPoint6[1676] = {X 275.5494, Y 85.6495, Z -8.0000, A 0.000, B 0.000, C 0.000 }
gfCNCPoint6[1677] = {X 262.6510, Y 80.5933, Z -8.0000, A 0.000, B 0.000, C 0.000 }
gfCNCPoint6[1678] = {X 237.8778, Y 96.6318, Z -8.0000, A 0.000, B 0.000, C 0.000 }
gfCNCPoint6[1679] = {X 237.8798, Y 97.0659, Z -8.0000, A 0.000, B 0.000, C 0.000 }
gfCNCPoint6[1680] = {X 237.8798, Y 98.0000, Z -8.0000, A 0.000, B 0.000, C 0.000 }
gfCNCPoint6[1681] = {X 237.7695, Y 98.9791, Z -8.0000, A 0.000, B 0.000, C 0.000 }
gfCNCPoint6[1682] = {X 237.4440, Y 99.9091, Z -8.0000, A 0.000, B 0.000, C 0.000 }
gfCNCPoint6[1683] = {X 236.9198, Y 100.7434, Z -8.0000, A 0.000, B 0.000, C 0.000 }
gfCNCPoint6[1684] = {X 236.2231, Y 101.4401, Z -8.0000, A 0.000, B 0.000, C 0.000 }
gfCNCPoint6[1685] = {X 235.3889, Y 101.9643, Z -8.0000, A 0.000, B 0.000, C 0.000 }
gfCNCPoint6[1686] = {X 234.4589, Y 102.2897, Z -8.0000, A 0.000, B 0.000, C 0.000 }
gfCNCPoint6[1687] = {X 233.4798, Y 102.4000, Z -8.0000, A 0.000, B 0.000, C 0.000 }
gfCNCPoint6[1688] = {X 214.1790, Y 102.4000, Z -8.0000, A 0.000, B 0.000, C 0.000 }
gfCNCPoint6[1689] = {X 213.7862, Y 102.3824, Z -8.0000, A 0.000, B 0.000, C 0.000 }
gfCNCPoint6[1690] = {X 213.3966, Y 102.3299, Z -8.0000, A 0.000, B 0.000, C 0.000 }
gfCNCPoint6[1691] = {X 213.0069, Y 102.3824, Z -8.0000, A 0.000, B 0.000, C 0.000 }
gfCNCPoint6[1692] = {X 212.6141, Y 102.4000, Z -8.0000, A 0.000, B 0.000, C 0.000 }
gfCNCPoint6[1693] = {X 194.9870, Y 102.4000, Z -8.0000, A 0.000, B 0.000, C 0.000 }
gfCNCPoint6[1694] = {X 194.0079, Y 102.2897, Z -8.0000, A 0.000, B 0.000, C 0.000 }
gfCNCPoint6[1695] = {X 193.0779, Y 101.9643, Z -8.0000, A 0.000, B 0.000, C 0.000 }
gfCNCPoint6[1696] = {X 192.2436, Y 101.4401, Z -8.0000, A 0.000, B 0.000, C 0.000 }
gfCNCPoint6[1697] = {X 191.5469, Y 100.7434, Z -8.0000, A 0.000, B 0.000, C 0.000 }
gfCNCPoint6[1698] = {X 191.0227, Y 99.9091, Z -8.0000, A 0.000, B 0.000, C 0.000 }
gfCNCPoint6[1699] = {X 190.6973, Y 98.9791, Z -8.0000, A 0.000, B 0.000, C 0.000 }
gfCNCPoint6[1700] = {X 190.5870, Y 98.0000, Z -8.0000, A 0.000, B 0.000, C 0.000 }
gfCNCPoint6[1701] = {X 190.5870, Y 97.0659, Z -8.0000, A 0.000, B 0.000, C 0.000 }
gfCNCPoint6[1702] = {X 190.6897, Y 96.1207, Z -8.0000, A 0.000, B 0.000, C 0.000 }
gfCNCPoint6[1703] = {X 190.9931, Y 95.2196, Z -8.0000, A 0.000, B 0.000, C 0.000 }
gfCNCPoint6[1704] = {X 191.4830, Y 94.4047, Z -8.0000, A 0.000, B 0.000, C 0.000 }
gfCNCPoint6[1705] = {X 188.5295, Y 91.1802, Z -8.0000, A 0.000, B 0.000, C 0.000 }
gfCNCPoint6[1706] = {X 150.1254, Y 91.1802, Z -8.0000, A 0.000, B 0.000, C 0.000 }
gfCNCPoint6[1707] = {X 147.2505, Y 94.3653, Z -8.0000, A 0.000, B 0.000, C 0.000 }
gfCNCPoint6[1708] = {X 147.7567, Y 95.1894, Z -8.0000, A 0.000, B 0.000, C 0.000 }
gfCNCPoint6[1709] = {X 148.0713, Y 96.1041, Z -8.0000, A 0.000, B 0.000, C 0.000 }
gfCNCPoint6[1710] = {X 148.1791, Y 97.0653, Z -8.0000, A 0.000, B 0.000, C 0.000 }
gfCNCPoint6[1711] = {X 148.1791, Y 98.0000, Z -8.0000, A 0.000, B 0.000, C 0.000 }
gfCNCPoint6[1712] = {X 148.0688, Y 98.9791, Z -8.0000, A 0.000, B 0.000, C 0.000 }
gfCNCPoint6[1713] = {X 147.7434, Y 99.9091, Z -8.0000, A 0.000, B 0.000, C 0.000 }
gfCNCPoint6[1714] = {X 147.2192, Y 100.7434, Z -8.0000, A 0.000, B 0.000, C 0.000 }
gfCNCPoint6[1715] = {X 146.5225, Y 101.4401, Z -8.0000, A 0.000, B 0.000, C 0.000 }
gfCNCPoint6[1716] = {X 145.6882, Y 101.9643, Z -8.0000, A 0.000, B 0.000, C 0.000 }
gfCNCPoint6[1717] = {X 144.7582, Y 102.2897, Z -8.0000, A 0.000, B 0.000, C 0.000 }
gfCNCPoint6[1718] = {X 143.7791, Y 102.4000, Z -8.0000, A 0.000, B 0.000, C 0.000 }
gfCNCPoint6[1719] = {X 125.0000, Y 102.4000, Z -8.0000, A 0.000, B 0.000, C 0.000 }
gfCNCPoint6[1720] = {X 124.0209, Y 102.2897, Z -8.0000, A 0.000, B 0.000, C 0.000 }
gfCNCPoint6[1721] = {X 123.0909, Y 101.9643, Z -8.0000, A 0.000, B 0.000, C 0.000 }
gfCNCPoint6[1722] = {X 122.2566, Y 101.4401, Z -8.0000, A 0.000, B 0.000, C 0.000 }
gfCNCPoint6[1723] = {X 121.5599, Y 100.7434, Z -8.0000, A 0.000, B 0.000, C 0.000 }
gfCNCPoint6[1724] = {X 121.0357, Y 99.9091, Z -8.0000, A 0.000, B 0.000, C 0.000 }
gfCNCPoint6[1725] = {X 120.7103, Y 98.9791, Z -8.0000, A 0.000, B 0.000, C 0.000 }
gfCNCPoint6[1726] = {X 120.6000, Y 98.0000, Z -8.0000, A 0.000, B 0.000, C 0.000 }
gfCNCPoint6[1727] = {X 120.6000, Y 97.0659, Z -8.0000, A 0.000, B 0.000, C 0.000 }
gfCNCPoint6[1728] = {X 120.7045, Y 96.1126, Z -8.0000, A 0.000, B 0.000, C 0.000 }
gfCNCPoint6[1729] = {X 121.0131, Y 95.2046, Z -8.0000, A 0.000, B 0.000, C 0.000 }
gfCNCPoint6[1730] = {X 121.5111, Y 94.3850, Z -8.0000, A 0.000, B 0.000, C 0.000 }
gfCNCPoint6[1731] = {X 122.1749, Y 93.6927, Z -8.0000, A 0.000, B 0.000, C 0.000 }
gfCNCPoint6[1732] = {X 122.9728, Y 93.1607, Z -8.0000, A 0.000, B 0.000, C 0.000 }
gfCNCPoint6[1733] = {X 123.8671, Y 92.8143, Z -8.0000, A 0.000, B 0.000, C 0.000 }
gfCNCPoint6[1734] = {X 124.8152, Y 92.6698, Z -8.0000, A 0.000, B 0.000, C 0.000 }
gfCNCPoint6[1735] = {X 124.8646, Y 92.6521, Z -8.0000, A 0.000, B 0.000, C 0.000 }
gfCNCPoint6[1736] = {X 124.9159, Y 92.6410, Z -8.0000, A 0.000, B 0.000, C 0.000 }
gfCNCPoint6[1737] = {X 125.4408, Y 92.5632, Z -8.0000, A 0.000, B 0.000, C 0.000 }
gfCNCPoint6[1738] = {X 126.2562, Y 92.4258, Z -8.0000, A 0.000, B 0.000, C 0.000 }
gfCNCPoint6[1739] = {X 127.0607, Y 92.2343, Z -8.0000, A 0.000, B 0.000, C 0.000 }
gfCNCPoint6[1740] = {X 128.2380, Y 91.1265, Z -8.0000, A 0.000, B 0.000, C 0.000 }
gfCNCPoint6[1741] = {X 129.3532, Y 89.9562, Z -8.0000, A 0.000, B 0.000, C 0.000 }
gfCNCPoint6[1742] = {X 155.5323, Y 61.2099, Z -8.0000, A 0.000, B 0.000, C 0.000 }
gfCNCPoint6[1743] = {X 155.1838, Y 60.4940, Z -8.0000, A 0.000, B 0.000, C 0.000 }
gfCNCPoint6[1744] = {X 154.9700, Y 59.7270, Z -8.0000, A 0.000, B 0.000, C 0.000 }
gfCNCPoint6[1745] = {X 154.8980, Y 58.9341, Z -8.0000, A 0.000, B 0.000, C 0.000 }
gfCNCPoint6[1746] = {X 154.8980, Y 58.0000, Z -8.0000, A 0.000, B 0.000, C 0.000 }
gfCNCPoint6[1747] = {X 155.0083, Y 57.0209, Z -8.0000, A 0.000, B 0.000, C 0.000 }
gfCNCPoint6[1748] = {X 155.3337, Y 56.0909, Z -8.0000, A 0.000, B 0.000, C 0.000 }
gfCNCPoint6[1749] = {X 155.8579, Y 55.2566, Z -8.0000, A 0.000, B 0.000, C 0.000 }
gfCNCPoint6[1750] = {X 156.5546, Y 54.5599, Z -8.0000, A 0.000, B 0.000, C 0.000 }
gfCNCPoint6[1751] = {X 157.3889, Y 54.0357, Z -8.0000, A 0.000, B 0.000, C 0.000 }
gfCNCPoint6[1752] = {X 158.3189, Y 53.7103, Z -8.0000, A 0.000, B 0.000, C 0.000 }
gfCNCPoint6[1753] = {X 159.2980, Y 53.6000, Z -8.0000, A 0.000, B 0.000, C 0.000 }
gfCNCPoint6[1754] = {X 178.5335, Y 53.6000, Z -8.0000, A 0.000, B 0.000, C 0.000 }
gfCNCPoint6[1755] = {X 179.5126, Y 53.7103, Z -8.0000, A 0.000, B 0.000, C 0.000 }
gfCNCPoint6[1756] = {X 180.4426, Y 54.0357, Z -8.0000, A 0.000, B 0.000, C 0.000 }
gfCNCPoint6[1757] = {X 181.2769, Y 54.5599, Z -8.0000, A 0.000, B 0.000, C 0.000 }
gfCNCPoint6[1758] = {X 181.9736, Y 55.2566, Z -8.0000, A 0.000, B 0.000, C 0.000 }
gfCNCPoint6[1759] = {X 182.4978, Y 56.0909, Z -8.0000, A 0.000, B 0.000, C 0.000 }
gfCNCPoint6[1760] = {X 182.8232, Y 57.0209, Z -8.0000, A 0.000, B 0.000, C 0.000 }
gfCNCPoint6[1761] = {X 182.9335, Y 58.0000, Z -8.0000, A 0.000, B 0.000, C 0.000 }
gfCNCPoint6[1762] = {X 182.9334, Y 58.9704, Z -8.0000, A 0.000, B 0.000, C 0.000 }
gfCNCPoint6[1763] = {X 182.8588, Y 59.7414, Z -8.0000, A 0.000, B 0.000, C 0.000 }
gfCNCPoint6[1764] = {X 182.6502, Y 60.4875, Z -8.0000, A 0.000, B 0.000, C 0.000 }
gfCNCPoint6[1765] = {X 182.3140, Y 61.1853, Z -8.0000, A 0.000, B 0.000, C 0.000 }
gfCNCPoint6[1766] = {X 209.3532, Y 90.7028, Z -8.0000, A 0.000, B 0.000, C 0.000 }
gfCNCPoint6[1767] = {X 210.0221, Y 91.3957, Z -8.0000, A 0.000, B 0.000, C 0.000 }
gfCNCPoint6[1768] = {X 210.7264, Y 92.0527, Z -8.0000, A 0.000, B 0.000, C 0.000 }
gfCNCPoint6[1769] = {X 211.1048, Y 92.3087, Z -8.0000, A 0.000, B 0.000, C 0.000 }
gfCNCPoint6[1770] = {X 211.5361, Y 92.4593, Z -8.0000, A 0.000, B 0.000, C 0.000 }
gfCNCPoint6[1771] = {X 212.1206, Y 92.5817, Z -8.0000, A 0.000, B 0.000, C 0.000 }
gfCNCPoint6[1772] = {X 213.3915, Y 92.7388, Z -8.0000, A 0.000, B 0.000, C 0.000 }
gfCNCPoint6[1773] = {X 214.4500, Y 92.6551, Z -8.0000, A 0.000, B 0.000, C 0.000 }
gfCNCPoint6[1774] = {X 215.5101, Y 92.5942, Z -8.0000, A 0.000, B 0.000, C 0.000 }
gfCNCPoint6[1775] = {X 216.1641, Y 92.5223, Z -8.0000, A 0.000, B 0.000, C 0.000 }
gfCNCPoint6[1776] = {X 216.7938, Y 92.3316, Z -8.0000, A 0.000, B 0.000, C 0.000 }
gfCNCPoint6[1777] = {X 217.3777, Y 92.0285, Z -8.0000, A 0.000, B 0.000, C 0.000 }
gfCNCPoint6[1778] = {X 222.9188, Y 88.4525, Z -8.0000, A 0.000, B 0.000, C 0.000 }
gfCNCPoint6[1779] = {X 245.6514, Y 73.9168, Z -8.0000, A 0.000, B 0.000, C 0.000 }
gfCNCPoint6[1780] = {X 221.6009, Y 64.4794, Z -8.0000, A 0.000, B 0.000, C 0.000 }
gfCNCPoint6[1781] = {X 219.8422, Y 63.8909, Z -8.0000, A 0.000, B 0.000, C 0.000 }
gfCNCPoint6[1782] = {X 218.0278, Y 63.5066, Z -8.0000, A 0.000, B 0.000, C 0.000 }
gfCNCPoint6[1783] = {X 216.1815, Y 63.3315, Z -8.0000, A 0.000, B 0.000, C 0.000 }
gfCNCPoint6[1784] = {X 215.2273, Y 63.1934, Z -8.0000, A 0.000, B 0.000, C 0.000 }
gfCNCPoint6[1785] = {X 214.3262, Y 62.8509, Z -8.0000, A 0.000, B 0.000, C 0.000 }
gfCNCPoint6[1786] = {X 213.5212, Y 62.3203, Z -8.0000, A 0.000, B 0.000, C 0.000 }
gfCNCPoint6[1787] = {X 212.8512, Y 61.6271, Z -8.0000, A 0.000, B 0.000, C 0.000 }
gfCNCPoint6[1788] = {X 212.3482, Y 60.8046, Z -8.0000, A 0.000, B 0.000, C 0.000 }
gfCNCPoint6[1789] = {X 212.0364, Y 59.8923, Z -8.0000, A 0.000, B 0.000, C 0.000 }
gfCNCPoint6[1790] = {X 211.9308, Y 58.9341, Z -8.0000, A 0.000, B 0.000, C 0.000 }
gfCNCPoint6[1791] = {X 211.9308, Y 58.0000, Z -8.0000, A 0.000, B 0.000, C 0.000 }
gfCNCPoint6[1792] = {X 212.0411, Y 57.0209, Z -8.0000, A 0.000, B 0.000, C 0.000 }
gfCNCPoint6[1793] = {X 212.3665, Y 56.0909, Z -8.0000, A 0.000, B 0.000, C 0.000 }
gfCNCPoint6[1794] = {X 212.8907, Y 55.2566, Z -8.0000, A 0.000, B 0.000, C 0.000 }
gfCNCPoint6[1795] = {X 213.5875, Y 54.5599, Z -8.0000, A 0.000, B 0.000, C 0.000 }
gfCNCPoint6[1796] = {X 214.4217, Y 54.0357, Z -8.0000, A 0.000, B 0.000, C 0.000 }
gfCNCPoint6[1797] = {X 215.3517, Y 53.7103, Z -8.0000, A 0.000, B 0.000, C 0.000 }
gfCNCPoint6[1798] = {X 216.3308, Y 53.6000, Z -8.0000, A 0.000, B 0.000, C 0.000 }
gfCNCPoint6[1799] = {X 237.2617, Y 53.6000, Z -8.0000, A 0.000, B 0.000, C 0.000 }
gfCNCPoint6[1800] = {X 238.2408, Y 53.7103, Z -8.0000, A 0.000, B 0.000, C 0.000 }
gfCNCPoint6[1801] = {X 239.1708, Y 54.0357, Z -8.0000, A 0.000, B 0.000, C 0.000 }
gfCNCPoint6[1802] = {X 240.0050, Y 54.5599, Z -8.0000, A 0.000, B 0.000, C 0.000 }
gfCNCPoint6[1803] = {X 240.7017, Y 55.2566, Z -8.0000, A 0.000, B 0.000, C 0.000 }
gfCNCPoint6[1804] = {X 241.2260, Y 56.0909, Z -8.0000, A 0.000, B 0.000, C 0.000 }
gfCNCPoint6[1805] = {X 241.5514, Y 57.0209, Z -8.0000, A 0.000, B 0.000, C 0.000 }
gfCNCPoint6[1806] = {X 241.6617, Y 58.0000, Z -8.0000, A 0.000, B 0.000, C 0.000 }
gfCNCPoint6[1807] = {X 241.6617, Y 58.1769, Z -8.0000, A 0.000, B 0.000, C 0.000 }
gfCNCPoint6[1808] = {X 248.1456, Y 60.7053, Z -8.0000, A 0.000, B 0.000, C 0.000 }
gfCNCPoint6[1809] = {X 275.5515, Y 71.5832, Z -8.0000, A 0.000, B 0.000, C 0.000 }
gfCNCPoint6[1810] = {X 275.5513, Y 63.2810, Z -8.0000, A 0.000, B 0.000, C 0.000 }
gfCNCPoint6[1811] = {X 274.6923, Y 63.0556, Z -8.0000, A 0.000, B 0.000, C 0.000 }
gfCNCPoint6[1812] = {X 273.8960, Y 62.6623, Z -8.0000, A 0.000, B 0.000, C 0.000 }
gfCNCPoint6[1813] = {X 273.1949, Y 62.1171, Z -8.0000, A 0.000, B 0.000, C 0.000 }
gfCNCPoint6[1814] = {X 272.6176, Y 61.4423, Z -8.0000, A 0.000, B 0.000, C 0.000 }
gfCNCPoint6[1815] = {X 272.1876, Y 60.6652, Z -8.0000, A 0.000, B 0.000, C 0.000 }
gfCNCPoint6[1816] = {X 271.9223, Y 59.8176, Z -8.0000, A 0.000, B 0.000, C 0.000 }
gfCNCPoint6[1817] = {X 271.8327, Y 58.9341, Z -8.0000, A 0.000, B 0.000, C 0.000 }
gfCNCPoint6[1818] = {X 271.8327, Y 58.0000, Z -8.0000, A 0.000, B 0.000, C 0.000 }
gfCNCPoint6[1819] = {X 271.9430, Y 57.0209, Z -8.0000, A 0.000, B 0.000, C 0.000 }
gfCNCPoint6[1820] = {X 272.2684, Y 56.0909, Z -8.0000, A 0.000, B 0.000, C 0.000 }
gfCNCPoint6[1821] = {X 272.7926, Y 55.2566, Z -8.0000, A 0.000, B 0.000, C 0.000 }
gfCNCPoint6[1822] = {X 273.4893, Y 54.5599, Z -8.0000, A 0.000, B 0.000, C 0.000 }
gfCNCPoint6[1823] = {X 274.3236, Y 54.0357, Z -8.0000, A 0.000, B 0.000, C 0.000 }
gfCNCPoint6[1824] = {X 275.2536, Y 53.7103, Z -8.0000, A 0.000, B 0.000, C 0.000 }
gfCNCPoint6[1825] = {X 276.2327, Y 53.6000, Z -8.0000, A 0.000, B 0.000, C 0.000 }
gfCNCPoint6[1826] = {X 292.7731, Y 53.6000, Z -8.0000, A 0.000, B 0.000, C 0.000 }
gfCNCPoint6[1827] = {X 293.7522, Y 53.7103, Z -8.0000, A 0.000, B 0.000, C 0.000 }
gfCNCPoint6[1828] = {X 294.6822, Y 54.0357, Z -8.0000, A 0.000, B 0.000, C 0.000 }
gfCNCPoint6[1829] = {X 295.5164, Y 54.5599, Z -8.0000, A 0.000, B 0.000, C 0.000 }
gfCNCPoint6[1830] = {X 296.2131, Y 55.2566, Z -8.0000, A 0.000, B 0.000, C 0.000 }
gfCNCPoint6[1831] = {X 296.7373, Y 56.0909, Z -8.0000, A 0.000, B 0.000, C 0.000 }
gfCNCPoint6[1832] = {X 297.0628, Y 57.0209, Z -8.0000, A 0.000, B 0.000, C 0.000 }
gfCNCPoint6[1833] = {X 297.1731, Y 58.0000, Z -8.0000, A 0.000, B 0.000, C 0.000 }
gfCNCPoint6[1834] = {X 297.1731, Y 58.9352, Z -8.0000, A 0.000, B 0.000, C 0.000 }
gfCNCPoint6[1835] = {X 297.0815, Y 59.8182, Z -8.0000, A 0.000, B 0.000, C 0.000 }
gfCNCPoint6[1836] = {X 296.8151, Y 60.6651, Z -8.0000, A 0.000, B 0.000, C 0.000 }
gfCNCPoint6[1837] = {X 296.3848, Y 61.4416, Z -8.0000, A 0.000, B 0.000, C 0.000 }
gfCNCPoint6[1838] = {X 295.8078, Y 62.1163, Z -8.0000, A 0.000, B 0.000, C 0.000 }
gfCNCPoint6[1839] = {X 295.1075, Y 62.6619, Z -8.0000, A 0.000, B 0.000, C 0.000 }
gfCNCPoint6[1840] = {X 294.3122, Y 63.0565, Z -8.0000, A 0.000, B 0.000, C 0.000 }
gfCNCPoint6[1841] = {X 293.4541, Y 63.2840, Z -8.0000, A 0.000, B 0.000, C 0.000 }
gfCNCPoint6[1842] = {X 293.4541, Y 92.7097, Z -8.0000, A 0.000, B 0.000, C 0.000 }
gfCNCPoint6[1843] = {X 294.3120, Y 92.9397, Z -8.0000, A 0.000, B 0.000, C 0.000 }
gfCNCPoint6[1844] = {X 295.1067, Y 93.3362, Z -8.0000, A 0.000, B 0.000, C 0.000 }
gfCNCPoint6[1845] = {X 295.8065, Y 93.8831, Z -8.0000, A 0.000, B 0.000, C 0.000 }
gfCNCPoint6[1846] = {X 296.3832, Y 94.5586, Z -8.0000, A 0.000, B 0.000, C 0.000 }
gfCNCPoint6[1847] = {X 296.8136, Y 95.3355, Z -8.0000, A 0.000, B 0.000, C 0.000 }
gfCNCPoint6[1848] = {X 297.0805, Y 96.1827, Z -8.0000, A 0.000, B 0.000, C 0.000 }
gfCNCPoint6[1849] = {X 297.1731, Y 97.0660, Z -8.0000, A 0.000, B 0.000, C 0.000 }
gfCNCPoint6[1850] = {X 297.1731, Y 97.6952, Z -8.0000, A 0.000, B 0.000, C 0.000 }
gfCNCPoint6[1851] = {X 297.6531, Y 97.6952, Z -8.0000, A 0.000, B 0.000, C 0.000 }
gfCNCPoint6[1852] = {X 314.2291, Y 97.6952, Z -8.0000, A 0.000, B 0.000, C 0.000 }
gfCNCPoint6[1853] = {X 313.3053, Y 97.0595, Z -8.0000, A 0.000, B 0.000, C 0.000 }
gfCNCPoint6[1854] = {X 312.4141, Y 96.3790, Z -8.0000, A 0.000, B 0.000, C 0.000 }
gfCNCPoint6[1855] = {X 311.1476, Y 95.2138, Z -8.0000, A 0.000, B 0.000, C 0.000 }
gfCNCPoint6[1856] = {X 310.0485, Y 93.8896, Z -8.0000, A 0.000, B 0.000, C 0.000 }
gfCNCPoint6[1857] = {X 309.2170, Y 92.5782, Z -8.0000, A 0.000, B 0.000, C 0.000 }
gfCNCPoint6[1858] = {X 308.5499, Y 91.1760, Z -8.0000, A 0.000, B 0.000, C 0.000 }
gfCNCPoint6[1859] = {X 307.9610, Y 89.2713, Z -8.0000, A 0.000, B 0.000, C 0.000 }
gfCNCPoint6[1860] = {X 307.5921, Y 87.3121, Z -8.0000, A 0.000, B 0.000, C 0.000 }
gfCNCPoint6[1861] = {X 307.4477, Y 85.3237, Z -8.0000, A 0.000, B 0.000, C 0.000 }
gfCNCPoint6[1862] = {X 307.4340, Y 84.6158, Z -8.0000, A 0.000, B 0.000, C 0.000 }
gfCNCPoint6[1863] = {X 307.4353, Y 63.6740, Z -8.0000, A 0.000, B 0.000, C 0.000 }
gfCNCPoint6[1864] = {X 306.4272, Y 63.3055, Z -8.0000, A 0.000, B 0.000, C 0.000 }
gfCNCPoint6[1865] = {X 305.5240, Y 62.7256, Z -8.0000, A 0.000, B 0.000, C 0.000 }
gfCNCPoint6[1866] = {X 304.7694, Y 61.9623, Z -8.0000, A 0.000, B 0.000, C 0.000 }
gfCNCPoint6[1867] = {X 304.2000, Y 61.0525, Z -8.0000, A 0.000, B 0.000, C 0.000 }
gfCNCPoint6[1868] = {X 303.8432, Y 60.0402, Z -8.0000, A 0.000, B 0.000, C 0.000 }
gfCNCPoint6[1869] = {X 303.7164, Y 58.9744, Z -8.0000, A 0.000, B 0.000, C 0.000 }
gfCNCPoint6[1870] = {X 303.7162, Y 58.0000, Z -8.0000, A 0.000, B 0.000, C 0.000 }
gfCNCPoint6[1871] = {X 303.8100, Y 57.0480, Z -8.0000, A 0.000, B 0.000, C 0.000 }
gfCNCPoint6[1872] = {X 304.0877, Y 56.1325, Z -8.0000, A 0.000, B 0.000, C 0.000 }
gfCNCPoint6[1873] = {X 304.5387, Y 55.2888, Z -8.0000, A 0.000, B 0.000, C 0.000 }
gfCNCPoint6[1874] = {X 305.1455, Y 54.5493, Z -8.0000, A 0.000, B 0.000, C 0.000 }
gfCNCPoint6[1875] = {X 305.8850, Y 53.9424, Z -8.0000, A 0.000, B 0.000, C 0.000 }
gfCNCPoint6[1876] = {X 306.7287, Y 53.4915, Z -8.0000, A 0.000, B 0.000, C 0.000 }
gfCNCPoint6[1877] = {X 307.6442, Y 53.2138, Z -8.0000, A 0.000, B 0.000, C 0.000 }
gfCNCPoint6[1878] = {X 308.5962, Y 53.1200, Z -8.0000, A 0.000, B 0.000, C 0.000 }
gfCNCPoint6[1879] = {X 324.3107, Y 53.1200, Z -8.0000, A 0.000, B 0.000, C 0.000 }
gfCNCPoint6[1880] = {X 325.2627, Y 53.2138, Z -8.0000, A 0.000, B 0.000, C 0.000 }
gfCNCPoint6[1881] = {X 326.1782, Y 53.4915, Z -8.0000, A 0.000, B 0.000, C 0.000 }
gfCNCPoint6[1882] = {X 327.0219, Y 53.9424, Z -8.0000, A 0.000, B 0.000, C 0.000 }
gfCNCPoint6[1883] = {X 327.7614, Y 54.5493, Z -8.0000, A 0.000, B 0.000, C 0.000 }
gfCNCPoint6[1884] = {X 328.3683, Y 55.2888, Z -8.0000, A 0.000, B 0.000, C 0.000 }
gfCNCPoint6[1885] = {X 328.8192, Y 56.1325, Z -8.0000, A 0.000, B 0.000, C 0.000 }
gfCNCPoint6[1886] = {X 329.0969, Y 57.0480, Z -8.0000, A 0.000, B 0.000, C 0.000 }
gfCNCPoint6[1887] = {X 329.1907, Y 58.0000, Z -8.0000, A 0.000, B 0.000, C 0.000 }
gfCNCPoint6[1888] = {X 329.1907, Y 58.9341, Z -8.0000, A 0.000, B 0.000, C 0.000 }
gfCNCPoint6[1889] = {X 329.0676, Y 60.0068, Z -8.0000, A 0.000, B 0.000, C 0.000 }
gfCNCPoint6[1890] = {X 328.7133, Y 61.0268, Z -8.0000, A 0.000, B 0.000, C 0.000 }
gfCNCPoint6[1891] = {X 328.1450, Y 61.9449, Z -8.0000, A 0.000, B 0.000, C 0.000 }
gfCNCPoint6[1892] = {X 327.3899, Y 62.7168, Z -8.0000, A 0.000, B 0.000, C 0.000 }
gfCNCPoint6[1893] = {X 326.4846, Y 63.3053, Z -8.0000, A 0.000, B 0.000, C 0.000 }
gfCNCPoint6[1894] = {X 325.4726, Y 63.6819, Z -8.0000, A 0.000, B 0.000, C 0.000 }
gfCNCPoint6[1895] = {X 325.4746, Y 83.2269, Z -8.0000, A 0.000, B 0.000, C 0.000 }
gfCNCPoint6[1896] = {X 325.4881, Y 84.6073, Z -8.0000, A 0.000, B 0.000, C 0.000 }
gfCNCPoint6[1897] = {X 325.5524, Y 85.7048, Z -8.0000, A 0.000, B 0.000, C 0.000 }
gfCNCPoint6[1898] = {X 325.7362, Y 86.7887, Z -8.0000, A 0.000, B 0.000, C 0.000 }
gfCNCPoint6[1899] = {X 326.0557, Y 87.0639, Z -8.0000, A 0.000, B 0.000, C 0.000 }
gfCNCPoint6[1900] = {X 326.4243, Y 87.2686, Z -8.0000, A 0.000, B 0.000, C 0.000 }
gfCNCPoint6[1901] = {X 328.1525, Y 87.9615, Z -8.0000, A 0.000, B 0.000, C 0.000 }
gfCNCPoint6[1902] = {X 329.9517, Y 88.4409, Z -8.0000, A 0.000, B 0.000, C 0.000 }
gfCNCPoint6[1903] = {X 333.0038, Y 88.9887, Z -8.0000, A 0.000, B 0.000, C 0.000 }
gfCNCPoint6[1904] = {X 336.0837, Y 89.3494, Z -8.0000, A 0.000, B 0.000, C 0.000 }
gfCNCPoint6[1905] = {X 340.4351, Y 89.6423, Z -8.0000, A 0.000, B 0.000, C 0.000 }
gfCNCPoint6[1906] = {X 344.7937, Y 89.7955, Z -8.0000, A 0.000, B 0.000, C 0.000 }
gfCNCPoint6[1907] = {X 349.1549, Y 89.8087, Z -8.0000, A 0.000, B 0.000, C 0.000 }
gfCNCPoint6[1908] = {X 353.2889, Y 89.7410, Z -8.0000, A 0.000, B 0.000, C 0.000 }
gfCNCPoint6[1909] = {X 357.4176, Y 89.5231, Z -8.0000, A 0.000, B 0.000, C 0.000 }
gfCNCPoint6[1910] = {X 361.5357, Y 89.1553, Z -8.0000, A 0.000, B 0.000, C 0.000 }
gfCNCPoint6[1911] = {X 363.5860, Y 88.8725, Z -8.0000, A 0.000, B 0.000, C 0.000 }
gfCNCPoint6[1912] = {X 365.6175, Y 88.4764, Z -8.0000, A 0.000, B 0.000, C 0.000 }
gfCNCPoint6[1913] = {X 367.6239, Y 87.9684, Z -8.0000, A 0.000, B 0.000, C 0.000 }
gfCNCPoint6[1914] = {X 368.9174, Y 87.4943, Z -8.0000, A 0.000, B 0.000, C 0.000 }
gfCNCPoint6[1915] = {X 370.1127, Y 86.8093, Z -8.0000, A 0.000, B 0.000, C 0.000 }
gfCNCPoint6[1916] = {X 370.2972, Y 85.3242, Z -8.0000, A 0.000, B 0.000, C 0.000 }
gfCNCPoint6[1917] = {X 370.3587, Y 83.8290, Z -8.0000, A 0.000, B 0.000, C 0.000 }
gfCNCPoint6[1918] = {X 370.3577, Y 63.6738, Z -8.0000, A 0.000, B 0.000, C 0.000 }
gfCNCPoint6[1919] = {X 369.3497, Y 63.3053, Z -8.0000, A 0.000, B 0.000, C 0.000 }
gfCNCPoint6[1920] = {X 368.4467, Y 62.7253, Z -8.0000, A 0.000, B 0.000, C 0.000 }
gfCNCPoint6[1921] = {X 367.6923, Y 61.9620, Z -8.0000, A 0.000, B 0.000, C 0.000 }
gfCNCPoint6[1922] = {X 367.1230, Y 61.0523, Z -8.0000, A 0.000, B 0.000, C 0.000 }
gfCNCPoint6[1923] = {X 366.7663, Y 60.0401, Z -8.0000, A 0.000, B 0.000, C 0.000 }
gfCNCPoint6[1924] = {X 366.6394, Y 58.9744, Z -8.0000, A 0.000, B 0.000, C 0.000 }
gfCNCPoint6[1925] = {X 366.6393, Y 58.0000, Z -8.0000, A 0.000, B 0.000, C 0.000 }
gfCNCPoint6[1926] = {X 366.7331, Y 57.0480, Z -8.0000, A 0.000, B 0.000, C 0.000 }
gfCNCPoint6[1927] = {X 367.0108, Y 56.1325, Z -8.0000, A 0.000, B 0.000, C 0.000 }
gfCNCPoint6[1928] = {X 367.4617, Y 55.2888, Z -8.0000, A 0.000, B 0.000, C 0.000 }
gfCNCPoint6[1929] = {X 368.0686, Y 54.5493, Z -8.0000, A 0.000, B 0.000, C 0.000 }
gfCNCPoint6[1930] = {X 368.8081, Y 53.9424, Z -8.0000, A 0.000, B 0.000, C 0.000 }
gfCNCPoint6[1931] = {X 369.6518, Y 53.4915, Z -8.0000, A 0.000, B 0.000, C 0.000 }
gfCNCPoint6[1932] = {X 370.5672, Y 53.2138, Z -8.0000, A 0.000, B 0.000, C 0.000 }
gfCNCPoint6[1933] = {X 371.5193, Y 53.1200, Z -8.0000, A 0.000, B 0.000, C 0.000 }
gfCNCPoint6[1934] = {X 388.0597, Y 53.1200, Z -8.0000, A 0.000, B 0.000, C 0.000 }
gfCNCPoint6[1935] = {X 389.0355, Y 53.2186, Z -8.0000, A 0.000, B 0.000, C 0.000 }
gfCNCPoint6[1936] = {X 389.9719, Y 53.5102, Z -8.0000, A 0.000, B 0.000, C 0.000 }
gfCNCPoint6[1937] = {X 390.8310, Y 53.9833, Z -8.0000, A 0.000, B 0.000, C 0.000 }
gfCNCPoint6[1938] = {X 391.5783, Y 54.6186, Z -8.0000, A 0.000, B 0.000, C 0.000 }
gfCNCPoint6[1939] = {X 392.1572, Y 55.3496, Z -8.0000, A 0.000, B 0.000, C 0.000 }
gfCNCPoint6[1940] = {X 392.5865, Y 56.1774, Z -8.0000, A 0.000, B 0.000, C 0.000 }
gfCNCPoint6[1941] = {X 392.8506, Y 57.0718, Z -8.0000, A 0.000, B 0.000, C 0.000 }
gfCNCPoint6[1942] = {X 392.9397, Y 58.0000, Z -8.0000, A 0.000, B 0.000, C 0.000 }
gfCNCPoint6[1943] = {X 392.9395, Y 58.9744, Z -8.0000, A 0.000, B 0.000, C 0.000 }
gfCNCPoint6[1944] = {X 392.8144, Y 60.0326, Z -8.0000, A 0.000, B 0.000, C 0.000 }
gfCNCPoint6[1945] = {X 392.4627, Y 61.0384, Z -8.0000, A 0.000, B 0.000, C 0.000 }
gfCNCPoint6[1946] = {X 392.0711, Y 61.7136, Z -8.0000, A 0.000, B 0.000, C 0.000 }
gfCNCPoint6[1947] = {X 391.5774, Y 62.3181, Z -8.0000, A 0.000, B 0.000, C 0.000 }
gfCNCPoint6[1948] = {X 390.8822, Y 62.9186, Z -8.0000, A 0.000, B 0.000, C 0.000 }
gfCNCPoint6[1949] = {X 390.0872, Y 63.3790, Z -8.0000, A 0.000, B 0.000, C 0.000 }
gfCNCPoint6[1950] = {X 389.2203, Y 63.6829, Z -8.0000, A 0.000, B 0.000, C 0.000 }
gfCNCPoint6[1951] = {X 389.2194, Y 73.4829, Z -8.0000, A 0.000, B 0.000, C 0.000 }
gfCNCPoint6[1952] = {X 398.8194, Y 73.4839, Z -8.0000, A 0.000, B 0.000, C 0.000 }
gfCNCPoint6[1953] = {X 398.8187, Y 80.5558, Z -8.0000, A 0.000, B 0.000, C 0.000 }
gfCNCPoint6[1954] = {X 405.8016, Y 76.0838, Z -8.0000, A 0.000, B 0.000, C 0.000 }
gfCNCPoint6[1955] = {X 400.0400, Y 73.8234, Z -8.0000, A 0.000, B 0.000, C 0.000 }
gfCNCPoint6[1956] = {X 399.4384, Y 73.6222, Z -8.0000, A 0.000, B 0.000, C 0.000 }
gfCNCPoint6[1957] = {X 398.8194, Y 73.4839, Z -8.0000, A 0.000, B 0.000, C 0.000 }
gfCNCPoint6[1958] = {X 396.4194, Y 73.4836, Z -8.0000, A 0.000, B 0.000, C 0.000 }
gfCNCPoint6[1959] = {X 396.4183, Y 84.5897, Z -8.0000, A 0.000, B 0.000, C 0.000 }
gfCNCPoint6[1960] = {X 396.4182, Y 84.9430, Z -8.0000, A 0.000, B 0.000, C 0.000 }
gfCNCPoint6[1961] = {X 411.0576, Y 75.5678, Z -8.0000, A 0.000, B 0.000, C 0.000 }
gfCNCPoint6[1962] = {X 400.9177, Y 71.5897, Z -8.0000, A 0.000, B 0.000, C 0.000 }
gfCNCPoint6[1963] = {X 399.6191, Y 71.1951, Z -8.0000, A 0.000, B 0.000, C 0.000 }
gfCNCPoint6[1964] = {X 398.2745, Y 71.0107, Z -8.0000, A 0.000, B 0.000, C 0.000 }
gfCNCPoint6[1965] = {X 397.3434, Y 70.9529, Z -8.0000, A 0.000, B 0.000, C 0.000 }
gfCNCPoint6[1966] = {X 396.4196, Y 70.8233, Z -8.0000, A 0.000, B 0.000, C 0.000 }
gfCNCPoint6[1967] = {X 396.4194, Y 73.4836, Z -8.0000, A 0.000, B 0.000, C 0.000 }
gfCNCPoint6[1968] = {X 394.0194, Y 73.4834, Z -8.0000, A 0.000, B 0.000, C 0.000 }
gfCNCPoint6[1969] = {X 394.0183, Y 84.5974, Z -8.0000, A 0.000, B 0.000, C 0.000 }
gfCNCPoint6[1970] = {X 394.0188, Y 84.7619, Z -8.0000, A 0.000, B 0.000, C 0.000 }
gfCNCPoint6[1971] = {X 394.0182, Y 84.9265, Z -8.0000, A 0.000, B 0.000, C 0.000 }
gfCNCPoint6[1972] = {X 393.9679, Y 86.3324, Z -8.0000, A 0.000, B 0.000, C 0.000 }
gfCNCPoint6[1973] = {X 393.8365, Y 87.7332, Z -8.0000, A 0.000, B 0.000, C 0.000 }
gfCNCPoint6[1974] = {X 395.0630, Y 87.4795, Z -8.0000, A 0.000, B 0.000, C 0.000 }
gfCNCPoint6[1975] = {X 396.3120, Y 87.3864, Z -8.0000, A 0.000, B 0.000, C 0.000 }
gfCNCPoint6[1976] = {X 396.7153, Y 87.3714, Z -8.0000, A 0.000, B 0.000, C 0.000 }
gfCNCPoint6[1977] = {X 397.1180, Y 87.3448, Z -8.0000, A 0.000, B 0.000, C 0.000 }
gfCNCPoint6[1978] = {X 416.3137, Y 75.0517, Z -8.0000, A 0.000, B 0.000, C 0.000 }
gfCNCPoint6[1979] = {X 401.7955, Y 69.3560, Z -8.0000, A 0.000, B 0.000, C 0.000 }
gfCNCPoint6[1980] = {X 400.6812, Y 68.9857, Z -8.0000, A 0.000, B 0.000, C 0.000 }
gfCNCPoint6[1981] = {X 399.5337, Y 68.7368, Z -8.0000, A 0.000, B 0.000, C 0.000 }
gfCNCPoint6[1982] = {X 398.3661, Y 68.6122, Z -8.0000, A 0.000, B 0.000, C 0.000 }
gfCNCPoint6[1983] = {X 397.6023, Y 68.5668, Z -8.0000, A 0.000, B 0.000, C 0.000 }
gfCNCPoint6[1984] = {X 396.8444, Y 68.4612, Z -8.0000, A 0.000, B 0.000, C 0.000 }
gfCNCPoint6[1985] = {X 395.3942, Y 68.0826, Z -8.0000, A 0.000, B 0.000, C 0.000 }
gfCNCPoint6[1986] = {X 394.0199, Y 67.4846, Z -8.0000, A 0.000, B 0.000, C 0.000 }
gfCNCPoint6[1987] = {X 394.0194, Y 73.4834, Z -8.0000, A 0.000, B 0.000, C 0.000 }
gfCNCPoint6[1988] = {X 391.6194, Y 73.4832, Z -8.0000, A 0.000, B 0.000, C 0.000 }
gfCNCPoint6[1989] = {X 391.6183, Y 84.6054, Z -8.0000, A 0.000, B 0.000, C 0.000 }
gfCNCPoint6[1990] = {X 391.5822, Y 86.0254, Z -8.0000, A 0.000, B 0.000, C 0.000 }
gfCNCPoint6[1991] = {X 391.4545, Y 87.4402, Z -8.0000, A 0.000, B 0.000, C 0.000 }
gfCNCPoint6[1992] = {X 391.2301, Y 88.8723, Z -8.0000, A 0.000, B 0.000, C 0.000 }
gfCNCPoint6[1993] = {X 390.9118, Y 90.2866, Z -8.0000, A 0.000, B 0.000, C 0.000 }
gfCNCPoint6[1994] = {X 390.3352, Y 92.0503, Z -8.0000, A 0.000, B 0.000, C 0.000 }
gfCNCPoint6[1995] = {X 389.5434, Y 93.7286, Z -8.0000, A 0.000, B 0.000, C 0.000 }
gfCNCPoint6[1996] = {X 388.5489, Y 95.2952, Z -8.0000, A 0.000, B 0.000, C 0.000 }
gfCNCPoint6[1997] = {X 389.3446, Y 95.2952, Z -8.0000, A 0.000, B 0.000, C 0.000 }
gfCNCPoint6[1998] = {X 389.7639, Y 94.0856, Z -8.0000, A 0.000, B 0.000, C 0.000 }
gfCNCPoint6[1999] = {X 390.3887, Y 92.9683, Z -8.0000, A 0.000, B 0.000, C 0.000 }
gfCNCPoint6[2000] = {X 391.1995, Y 91.9776, Z -8.0000, A 0.000, B 0.000, C 0.000 }
gfCNCPoint6[2001] = {X 392.1713, Y 91.1443, Z -8.0000, A 0.000, B 0.000, C 0.000 }
gfCNCPoint6[2002] = {X 393.2740, Y 90.4941, Z -8.0000, A 0.000, B 0.000, C 0.000 }
gfCNCPoint6[2003] = {X 394.4736, Y 90.0471, Z -8.0000, A 0.000, B 0.000, C 0.000 }
gfCNCPoint6[2004] = {X 395.4029, Y 89.8554, Z -8.0000, A 0.000, B 0.000, C 0.000 }
gfCNCPoint6[2005] = {X 396.3493, Y 89.7862, Z -8.0000, A 0.000, B 0.000, C 0.000 }
gfCNCPoint6[2006] = {X 397.1455, Y 89.7469, Z -8.0000, A 0.000, B 0.000, C 0.000 }
gfCNCPoint6[2007] = {X 397.9389, Y 89.6690, Z -8.0000, A 0.000, B 0.000, C 0.000 }
gfCNCPoint6[2008] = {X 421.5697, Y 74.5357, Z -8.0000, A 0.000, B 0.000, C 0.000 }
gfCNCPoint6[2009] = {X 402.6732, Y 67.1222, Z -8.0000, A 0.000, B 0.000, C 0.000 }
gfCNCPoint6[2010] = {X 401.3006, Y 66.6670, Z -8.0000, A 0.000, B 0.000, C 0.000 }
gfCNCPoint6[2011] = {X 399.8868, Y 66.3628, Z -8.0000, A 0.000, B 0.000, C 0.000 }
gfCNCPoint6[2012] = {X 398.4484, Y 66.2132, Z -8.0000, A 0.000, B 0.000, C 0.000 }
gfCNCPoint6[2013] = {X 397.3043, Y 66.1054, Z -8.0000, A 0.000, B 0.000, C 0.000 }
gfCNCPoint6[2014] = {X 396.1914, Y 65.8188, Z -8.0000, A 0.000, B 0.000, C 0.000 }
gfCNCPoint6[2015] = {X 395.1375, Y 65.3606, Z -8.0000, A 0.000, B 0.000, C 0.000 }
gfCNCPoint6[2016] = {X 394.1688, Y 64.7423, Z -8.0000, A 0.000, B 0.000, C 0.000 }
gfCNCPoint6[2017] = {X 393.3095, Y 63.9793, Z -8.0000, A 0.000, B 0.000, C 0.000 }
gfCNCPoint6[2018] = {X 392.5130, Y 64.6963, Z -8.0000, A 0.000, B 0.000, C 0.000 }
gfCNCPoint6[2019] = {X 391.6201, Y 65.2889, Z -8.0000, A 0.000, B 0.000, C 0.000 }
gfCNCPoint6[2020] = {X 391.6194, Y 73.4832, Z -8.0000, A 0.000, B 0.000, C 0.000 }
gfCNCPoint6[2021] = {X 389.2194, Y 73.4829, Z -8.0000, A 0.000, B 0.000, C 0.000 }
gfCNCPoint6[2022] = {X 389.2183, Y 84.6139, Z -8.0000, A 0.000, B 0.000, C 0.000 }
gfCNCPoint6[2023] = {X 389.1564, Y 86.3199, Z -8.0000, A 0.000, B 0.000, C 0.000 }
gfCNCPoint6[2024] = {X 388.9460, Y 88.0140, Z -8.0000, A 0.000, B 0.000, C 0.000 }
gfCNCPoint6[2025] = {X 388.5888, Y 89.6833, Z -8.0000, A 0.000, B 0.000, C 0.000 }
gfCNCPoint6[2026] = {X 388.1052, Y 91.1630, Z -8.0000, A 0.000, B 0.000, C 0.000 }
gfCNCPoint6[2027] = {X 387.4411, Y 92.5708, Z -8.0000, A 0.000, B 0.000, C 0.000 }
gfCNCPoint6[2028] = {X 386.6069, Y 93.8850, Z -8.0000, A 0.000, B 0.000, C 0.000 }
gfCNCPoint6[2029] = {X 385.8874, Y 94.7853, Z -8.0000, A 0.000, B 0.000, C 0.000 }
gfCNCPoint6[2030] = {X 385.0880, Y 95.6153, Z -8.0000, A 0.000, B 0.000, C 0.000 }
gfCNCPoint6[2031] = {X 383.8166, Y 96.7132, Z -8.0000, A 0.000, B 0.000, C 0.000 }
gfCNCPoint6[2032] = {X 382.4538, Y 97.6952, Z -8.0000, A 0.000, B 0.000, C 0.000 }
gfCNCPoint6[2033] = {X 382.1905, Y 97.2938, Z -8.0000, A 0.000, B 0.000, C 0.000 }
gfCNCPoint6[2034] = {X 381.0215, Y 98.0005, Z -8.0000, A 0.000, B 0.000, C 0.000 }
gfCNCPoint6[2035] = {X 379.8038, Y 98.6196, Z -8.0000, A 0.000, B 0.000, C 0.000 }
gfCNCPoint6[2036] = {X 377.5266, Y 99.5769, Z -8.0000, A 0.000, B 0.000, C 0.000 }
gfCNCPoint6[2037] = {X 375.1868, Y 100.3690, Z -8.0000, A 0.000, B 0.000, C 0.000 }
gfCNCPoint6[2038] = {X 372.7964, Y 100.9920, Z -8.0000, A 0.000, B 0.000, C 0.000 }
gfCNCPoint6[2039] = {X 369.1114, Y 101.7090, Z -8.0000, A 0.000, B 0.000, C 0.000 }
gfCNCPoint6[2040] = {X 365.3967, Y 102.2516, Z -8.0000, A 0.000, B 0.000, C 0.000 }
gfCNCPoint6[2041] = {X 361.6605, Y 102.6187, Z -8.0000, A 0.000, B 0.000, C 0.000 }
gfCNCPoint6[2042] = {X 355.4196, Y 102.9718, Z -8.0000, A 0.000, B 0.000, C 0.000 }
gfCNCPoint6[2043] = {X 349.1703, Y 103.1106, Z -8.0000, A 0.000, B 0.000, C 0.000 }
gfCNCPoint6[2044] = {X 342.9199, Y 103.0347, Z -8.0000, A 0.000, B 0.000, C 0.000 }
gfCNCPoint6[2045] = {X 342.3911, Y 103.0160, Z -8.0000, A 0.000, B 0.000, C 0.000 }
gfCNCPoint6[2046] = {X 342.2333, Y 103.0136, Z -8.0000, A 0.000, B 0.000, C 0.000 }
gfCNCPoint6[2047] = {X 337.5864, Y 102.8233, Z -8.0000, A 0.000, B 0.000, C 0.000 }
gfCNCPoint6[2048] = {X 332.9511, Y 102.4430, Z -8.0000, A 0.000, B 0.000, C 0.000 }
gfCNCPoint6[2049] = {X 328.3353, Y 101.8734, Z -8.0000, A 0.000, B 0.000, C 0.000 }
gfCNCPoint6[2050] = {X 325.2612, Y 101.3340, Z -8.0000, A 0.000, B 0.000, C 0.000 }
gfCNCPoint6[2051] = {X 322.2303, Y 100.5892, Z -8.0000, A 0.000, B 0.000, C 0.000 }
gfCNCPoint6[2052] = {X 319.2562, Y 99.6425, Z -8.0000, A 0.000, B 0.000, C 0.000 }
gfCNCPoint6[2053] = {X 317.5110, Y 98.9444, Z -8.0000, A 0.000, B 0.000, C 0.000 }
gfCNCPoint6[2054] = {X 315.8311, Y 98.1012, Z -8.0000, A 0.000, B 0.000, C 0.000 }
gfCNCPoint6[2055] = {X 314.2285, Y 97.1190, Z -8.0000, A 0.000, B 0.000, C 0.000 }
gfCNCPoint6[2056] = {X 312.7147, Y 96.0048, Z -8.0000, A 0.000, B 0.000, C 0.000 }
gfCNCPoint6[2057] = {X 311.5497, Y 94.9397, Z -8.0000, A 0.000, B 0.000, C 0.000 }
gfCNCPoint6[2058] = {X 310.5301, Y 93.7348, Z -8.0000, A 0.000, B 0.000, C 0.000 }
gfCNCPoint6[2059] = {X 309.6725, Y 92.4096, Z -8.0000, A 0.000, B 0.000, C 0.000 }
gfCNCPoint6[2060] = {X 308.9910, Y 90.9859, Z -8.0000, A 0.000, B 0.000, C 0.000 }
gfCNCPoint6[2061] = {X 308.4228, Y 89.1399, Z -8.0000, A 0.000, B 0.000, C 0.000 }
gfCNCPoint6[2062] = {X 308.0668, Y 87.2416, Z -8.0000, A 0.000, B 0.000, C 0.000 }
gfCNCPoint6[2063] = {X 307.9276, Y 85.3153, Z -8.0000, A 0.000, B 0.000, C 0.000 }
gfCNCPoint6[2064] = {X 307.9140, Y 84.6159, Z -8.0000, A 0.000, B 0.000, C 0.000 }
gfCNCPoint6[2065] = {X 307.9153, Y 63.2811, Z -8.0000, A 0.000, B 0.000, C 0.000 }
gfCNCPoint6[2066] = {X 307.0562, Y 63.0557, Z -8.0000, A 0.000, B 0.000, C 0.000 }
gfCNCPoint6[2067] = {X 306.2598, Y 62.6625, Z -8.0000, A 0.000, B 0.000, C 0.000 }
gfCNCPoint6[2068] = {X 305.5586, Y 62.1173, Z -8.0000, A 0.000, B 0.000, C 0.000 }
gfCNCPoint6[2069] = {X 304.9812, Y 61.4424, Z -8.0000, A 0.000, B 0.000, C 0.000 }
gfCNCPoint6[2070] = {X 304.5511, Y 60.6653, Z -8.0000, A 0.000, B 0.000, C 0.000 }
gfCNCPoint6[2071] = {X 304.2859, Y 59.8177, Z -8.0000, A 0.000, B 0.000, C 0.000 }
gfCNCPoint6[2072] = {X 304.1962, Y 58.9341, Z -8.0000, A 0.000, B 0.000, C 0.000 }
gfCNCPoint6[2073] = {X 304.1962, Y 58.0000, Z -8.0000, A 0.000, B 0.000, C 0.000 }
gfCNCPoint6[2074] = {X 304.3065, Y 57.0209, Z -8.0000, A 0.000, B 0.000, C 0.000 }
gfCNCPoint6[2075] = {X 304.6320, Y 56.0909, Z -8.0000, A 0.000, B 0.000, C 0.000 }
gfCNCPoint6[2076] = {X 305.1562, Y 55.2566, Z -8.0000, A 0.000, B 0.000, C 0.000 }
gfCNCPoint6[2077] = {X 305.8529, Y 54.5599, Z -8.0000, A 0.000, B 0.000, C 0.000 }
gfCNCPoint6[2078] = {X 306.6871, Y 54.0357, Z -8.0000, A 0.000, B 0.000, C 0.000 }
gfCNCPoint6[2079] = {X 307.6171, Y 53.7103, Z -8.0000, A 0.000, B 0.000, C 0.000 }
gfCNCPoint6[2080] = {X 308.5962, Y 53.6000, Z -8.0000, A 0.000, B 0.000, C 0.000 }
gfCNCPoint6[2081] = {X 324.3107, Y 53.6000, Z -8.0000, A 0.000, B 0.000, C 0.000 }
gfCNCPoint6[2082] = {X 325.2898, Y 53.7103, Z -8.0000, A 0.000, B 0.000, C 0.000 }
gfCNCPoint6[2083] = {X 326.2198, Y 54.0357, Z -8.0000, A 0.000, B 0.000, C 0.000 }
gfCNCPoint6[2084] = {X 327.0540, Y 54.5599, Z -8.0000, A 0.000, B 0.000, C 0.000 }
gfCNCPoint6[2085] = {X 327.7507, Y 55.2566, Z -8.0000, A 0.000, B 0.000, C 0.000 }
gfCNCPoint6[2086] = {X 328.2750, Y 56.0909, Z -8.0000, A 0.000, B 0.000, C 0.000 }
gfCNCPoint6[2087] = {X 328.6004, Y 57.0209, Z -8.0000, A 0.000, B 0.000, C 0.000 }
gfCNCPoint6[2088] = {X 328.7107, Y 58.0000, Z -8.0000, A 0.000, B 0.000, C 0.000 }
gfCNCPoint6[2089] = {X 328.7107, Y 58.9361, Z -8.0000, A 0.000, B 0.000, C 0.000 }
gfCNCPoint6[2090] = {X 328.6173, Y 59.8190, Z -8.0000, A 0.000, B 0.000, C 0.000 }
gfCNCPoint6[2091] = {X 328.3501, Y 60.6656, Z -8.0000, A 0.000, B 0.000, C 0.000 }
gfCNCPoint6[2092] = {X 327.9197, Y 61.4420, Z -8.0000, A 0.000, B 0.000, C 0.000 }
gfCNCPoint6[2093] = {X 327.3433, Y 62.1172, Z -8.0000, A 0.000, B 0.000, C 0.000 }
gfCNCPoint6[2094] = {X 326.6440, Y 62.6642, Z -8.0000, A 0.000, B 0.000, C 0.000 }
gfCNCPoint6[2095] = {X 325.8499, Y 63.0610, Z -8.0000, A 0.000, B 0.000, C 0.000 }
gfCNCPoint6[2096] = {X 324.9926, Y 63.2917, Z -8.0000, A 0.000, B 0.000, C 0.000 }
gfCNCPoint6[2097] = {X 324.9946, Y 83.2293, Z -8.0000, A 0.000, B 0.000, C 0.000 }
gfCNCPoint6[2098] = {X 325.0081, Y 84.6141, Z -8.0000, A 0.000, B 0.000, C 0.000 }
gfCNCPoint6[2099] = {X 325.0831, Y 85.8239, Z -8.0000, A 0.000, B 0.000, C 0.000 }
gfCNCPoint6[2100] = {X 325.2965, Y 87.0170, Z -8.0000, A 0.000, B 0.000, C 0.000 }
gfCNCPoint6[2101] = {X 325.7312, Y 87.4221, Z -8.0000, A 0.000, B 0.000, C 0.000 }
gfCNCPoint6[2102] = {X 326.2480, Y 87.7156, Z -8.0000, A 0.000, B 0.000, C 0.000 }
gfCNCPoint6[2103] = {X 328.0177, Y 88.4223, Z -8.0000, A 0.000, B 0.000, C 0.000 }
gfCNCPoint6[2104] = {X 329.8594, Y 88.9120, Z -8.0000, A 0.000, B 0.000, C 0.000 }
gfCNCPoint6[2105] = {X 332.9373, Y 89.4641, Z -8.0000, A 0.000, B 0.000, C 0.000 }
gfCNCPoint6[2106] = {X 336.0431, Y 89.8276, Z -8.0000, A 0.000, B 0.000, C 0.000 }
gfCNCPoint6[2107] = {X 340.4120, Y 90.1218, Z -8.0000, A 0.000, B 0.000, C 0.000 }
gfCNCPoint6[2108] = {X 344.7882, Y 90.2755, Z -8.0000, A 0.000, B 0.000, C 0.000 }
gfCNCPoint6[2109] = {X 349.1670, Y 90.2886, Z -8.0000, A 0.000, B 0.000, C 0.000 }
gfCNCPoint6[2110] = {X 353.3143, Y 90.2203, Z -8.0000, A 0.000, B 0.000, C 0.000 }
gfCNCPoint6[2111] = {X 357.4564, Y 90.0015, Z -8.0000, A 0.000, B 0.000, C 0.000 }
gfCNCPoint6[2112] = {X 361.5878, Y 89.6325, Z -8.0000, A 0.000, B 0.000, C 0.000 }
gfCNCPoint6[2113] = {X 363.6656, Y 89.3458, Z -8.0000, A 0.000, B 0.000, C 0.000 }
gfCNCPoint6[2114] = {X 365.7243, Y 88.9444, Z -8.0000, A 0.000, B 0.000, C 0.000 }
gfCNCPoint6[2115] = {X 367.7576, Y 88.4294, Z -8.0000, A 0.000, B 0.000, C 0.000 }
gfCNCPoint6[2116] = {X 368.6806, Y 88.1194, Z -8.0000, A 0.000, B 0.000, C 0.000 }
gfCNCPoint6[2117] = {X 369.5628, Y 87.7075, Z -8.0000, A 0.000, B 0.000, C 0.000 }
gfCNCPoint6[2118] = {X 370.3930, Y 87.1990, Z -8.0000, A 0.000, B 0.000, C 0.000 }
gfCNCPoint6[2119] = {X 370.5195, Y 87.0672, Z -8.0000, A 0.000, B 0.000, C 0.000 }
gfCNCPoint6[2120] = {X 370.5848, Y 86.8966, Z -8.0000, A 0.000, B 0.000, C 0.000 }
gfCNCPoint6[2121] = {X 370.7752, Y 85.3681, Z -8.0000, A 0.000, B 0.000, C 0.000 }
gfCNCPoint6[2122] = {X 370.8387, Y 83.8290, Z -8.0000, A 0.000, B 0.000, C 0.000 }
gfCNCPoint6[2123] = {X 370.8376, Y 63.2809, Z -8.0000, A 0.000, B 0.000, C 0.000 }
gfCNCPoint6[2124] = {X 369.9786, Y 63.0555, Z -8.0000, A 0.000, B 0.000, C 0.000 }
gfCNCPoint6[2125] = {X 369.1824, Y 62.6622, Z -8.0000, A 0.000, B 0.000, C 0.000 }
gfCNCPoint6[2126] = {X 368.4814, Y 62.1170, Z -8.0000, A 0.000, B 0.000, C 0.000 }
gfCNCPoint6[2127] = {X 367.9041, Y 61.4422, Z -8.0000, A 0.000, B 0.000, C 0.000 }
gfCNCPoint6[2128] = {X 367.4741, Y 60.6651, Z -8.0000, A 0.000, B 0.000, C 0.000 }
gfCNCPoint6[2129] = {X 367.2089, Y 59.8176, Z -8.0000, A 0.000, B 0.000, C 0.000 }
gfCNCPoint6[2130] = {X 367.1193, Y 58.9341, Z -8.0000, A 0.000, B 0.000, C 0.000 }
gfCNCPoint6[2131] = {X 367.1193, Y 58.0000, Z -8.0000, A 0.000, B 0.000, C 0.000 }
gfCNCPoint6[2132] = {X 367.2296, Y 57.0209, Z -8.0000, A 0.000, B 0.000, C 0.000 }
gfCNCPoint6[2133] = {X 367.5550, Y 56.0909, Z -8.0000, A 0.000, B 0.000, C 0.000 }
gfCNCPoint6[2134] = {X 368.0792, Y 55.2566, Z -8.0000, A 0.000, B 0.000, C 0.000 }
gfCNCPoint6[2135] = {X 368.7759, Y 54.5599, Z -8.0000, A 0.000, B 0.000, C 0.000 }
gfCNCPoint6[2136] = {X 369.6102, Y 54.0357, Z -8.0000, A 0.000, B 0.000, C 0.000 }
gfCNCPoint6[2137] = {X 370.5402, Y 53.7103, Z -8.0000, A 0.000, B 0.000, C 0.000 }
gfCNCPoint6[2138] = {X 371.5193, Y 53.6000, Z -8.0000, A 0.000, B 0.000, C 0.000 }
gfCNCPoint6[2139] = {X 388.0597, Y 53.6000, Z -8.0000, A 0.000, B 0.000, C 0.000 }
gfCNCPoint6[2140] = {X 389.0388, Y 53.7103, Z -8.0000, A 0.000, B 0.000, C 0.000 }
gfCNCPoint6[2141] = {X 389.9688, Y 54.0357, Z -8.0000, A 0.000, B 0.000, C 0.000 }
gfCNCPoint6[2142] = {X 390.8030, Y 54.5599, Z -8.0000, A 0.000, B 0.000, C 0.000 }
gfCNCPoint6[2143] = {X 391.4997, Y 55.2566, Z -8.0000, A 0.000, B 0.000, C 0.000 }
gfCNCPoint6[2144] = {X 392.0239, Y 56.0909, Z -8.0000, A 0.000, B 0.000, C 0.000 }
gfCNCPoint6[2145] = {X 392.3494, Y 57.0209, Z -8.0000, A 0.000, B 0.000, C 0.000 }
gfCNCPoint6[2146] = {X 392.4597, Y 58.0000, Z -8.0000, A 0.000, B 0.000, C 0.000 }
gfCNCPoint6[2147] = {X 392.4595, Y 58.9704, Z -8.0000, A 0.000, B 0.000, C 0.000 }
gfCNCPoint6[2148] = {X 392.3468, Y 59.9245, Z -8.0000, A 0.000, B 0.000, C 0.000 }
gfCNCPoint6[2149] = {X 392.0296, Y 60.8314, Z -8.0000, A 0.000, B 0.000, C 0.000 }
gfCNCPoint6[2150] = {X 391.5893, Y 61.5619, Z -8.0000, A 0.000, B 0.000, C 0.000 }
gfCNCPoint6[2151] = {X 391.0170, Y 62.1944, Z -8.0000, A 0.000, B 0.000, C 0.000 }
gfCNCPoint6[2152] = {X 390.3339, Y 62.7053, Z -8.0000, A 0.000, B 0.000, C 0.000 }
gfCNCPoint6[2153] = {X 389.5655, Y 63.0755, Z -8.0000, A 0.000, B 0.000, C 0.000 }
gfCNCPoint6[2154] = {X 388.7403, Y 63.2914, Z -8.0000, A 0.000, B 0.000, C 0.000 }
gfCNCPoint6[2155] = {X 388.7403, Y 83.9247, Z -8.0000, A 0.000, B 0.000, C 0.000 }
gfCNCPoint6[2156] = {X 388.7383, Y 84.6150, Z -8.0000, A 0.000, B 0.000, C 0.000 }
gfCNCPoint6[2157] = {X 388.6781, Y 86.2799, Z -8.0000, A 0.000, B 0.000, C 0.000 }
gfCNCPoint6[2158] = {X 388.4729, Y 87.9333, Z -8.0000, A 0.000, B 0.000, C 0.000 }
gfCNCPoint6[2159] = {X 388.1243, Y 89.5625, Z -8.0000, A 0.000, B 0.000, C 0.000 }
gfCNCPoint6[2160] = {X 387.5916, Y 91.1521, Z -8.0000, A 0.000, B 0.000, C 0.000 }
gfCNCPoint6[2161] = {X 386.8425, Y 92.6519, Z -8.0000, A 0.000, B 0.000, C 0.000 }
gfCNCPoint6[2162] = {X 385.8916, Y 94.0326, Z -8.0000, A 0.000, B 0.000, C 0.000 }
gfCNCPoint6[2163] = {X 384.7575, Y 95.2672, Z -8.0000, A 0.000, B 0.000, C 0.000 }
gfCNCPoint6[2164] = {X 383.5186, Y 96.3369, Z -8.0000, A 0.000, B 0.000, C 0.000 }
gfCNCPoint6[2165] = {X 382.1905, Y 97.2938, Z -8.0000, A 0.000, B 0.000, C 0.000 }
gfCNCPoint6[2166] = {X 382.4538, Y 97.6952, Z -8.0000, A 0.000, B 0.000, C 0.000 }
gfCNCPoint6[2167] = {X 391.5259, Y 97.6952, Z -8.0000, A 0.000, B 0.000, C 0.000 }
gfCNCPoint6[2168] = {X 391.5259, Y 97.0659, Z -8.0000, A 0.000, B 0.000, C 0.000 }
gfCNCPoint6[2169] = {X 391.6191, Y 96.1168, Z -8.0000, A 0.000, B 0.000, C 0.000 }
gfCNCPoint6[2170] = {X 391.8952, Y 95.2039, Z -8.0000, A 0.000, B 0.000, C 0.000 }
gfCNCPoint6[2171] = {X 392.3435, Y 94.3621, Z -8.0000, A 0.000, B 0.000, C 0.000 }
gfCNCPoint6[2172] = {X 392.9470, Y 93.6236, Z -8.0000, A 0.000, B 0.000, C 0.000 }
gfCNCPoint6[2173] = {X 393.6826, Y 93.0165, Z -8.0000, A 0.000, B 0.000, C 0.000 }
gfCNCPoint6[2174] = {X 394.5222, Y 92.5642, Z -8.0000, A 0.000, B 0.000, C 0.000 }
gfCNCPoint6[2175] = {X 395.4338, Y 92.2837, Z -8.0000, A 0.000, B 0.000, C 0.000 }
gfCNCPoint6[2176] = {X 396.3825, Y 92.1860, Z -8.0000, A 0.000, B 0.000, C 0.000 }
gfCNCPoint6[2177] = {X 397.3055, Y 92.1442, Z -8.0000, A 0.000, B 0.000, C 0.000 }
gfCNCPoint6[2178] = {X 398.2254, Y 92.0571, Z -8.0000, A 0.000, B 0.000, C 0.000 }
gfCNCPoint6[2179] = {X 398.7531, Y 91.9290, Z -8.0000, A 0.000, B 0.000, C 0.000 }
gfCNCPoint6[2180] = {X 399.2389, Y 91.6865, Z -8.0000, A 0.000, B 0.000, C 0.000 }
gfCNCPoint6[2181] = {X 426.8257, Y 74.0197, Z -8.0000, A 0.000, B 0.000, C 0.000 }
gfCNCPoint6[2182] = {X 403.5510, Y 64.8885, Z -8.0000, A 0.000, B 0.000, C 0.000 }
gfCNCPoint6[2183] = {X 401.9166, Y 64.3473, Z -8.0000, A 0.000, B 0.000, C 0.000 }
gfCNCPoint6[2184] = {X 400.2329, Y 63.9877, Z -8.0000, A 0.000, B 0.000, C 0.000 }
gfCNCPoint6[2185] = {X 398.5199, Y 63.8139, Z -8.0000, A 0.000, B 0.000, C 0.000 }
gfCNCPoint6[2186] = {X 397.5544, Y 63.7098, Z -8.0000, A 0.000, B 0.000, C 0.000 }
gfCNCPoint6[2187] = {X 396.6285, Y 63.4165, Z -8.0000, A 0.000, B 0.000, C 0.000 }
gfCNCPoint6[2188] = {X 395.7791, Y 62.9457, Z -8.0000, A 0.000, B 0.000, C 0.000 }
gfCNCPoint6[2189] = {X 395.0397, Y 62.3161, Z -8.0000, A 0.000, B 0.000, C 0.000 }
gfCNCPoint6[2190] = {X 394.4660, Y 61.5934, Z -8.0000, A 0.000, B 0.000, C 0.000 }
gfCNCPoint6[2191] = {X 394.0386, Y 60.7757, Z -8.0000, A 0.000, B 0.000, C 0.000 }
gfCNCPoint6[2192] = {X 393.7727, Y 59.8922, Z -8.0000, A 0.000, B 0.000, C 0.000 }
gfCNCPoint6[2193] = {X 393.6779, Y 58.9744, Z -8.0000, A 0.000, B 0.000, C 0.000 }
gfCNCPoint6[2194] = {X 393.6777, Y 58.0000, Z -8.0000, A 0.000, B 0.000, C 0.000 }
gfCNCPoint6[2195] = {X 393.7668, Y 57.0718, Z -8.0000, A 0.000, B 0.000, C 0.000 }
gfCNCPoint6[2196] = {X 394.0309, Y 56.1774, Z -8.0000, A 0.000, B 0.000, C 0.000 }
gfCNCPoint6[2197] = {X 394.4602, Y 55.3496, Z -8.0000, A 0.000, B 0.000, C 0.000 }
gfCNCPoint6[2198] = {X 395.0391, Y 54.6186, Z -8.0000, A 0.000, B 0.000, C 0.000 }
gfCNCPoint6[2199] = {X 395.7864, Y 53.9833, Z -8.0000, A 0.000, B 0.000, C 0.000 }
gfCNCPoint6[2200] = {X 396.6455, Y 53.5102, Z -8.0000, A 0.000, B 0.000, C 0.000 }
gfCNCPoint6[2201] = {X 397.5819, Y 53.2186, Z -8.0000, A 0.000, B 0.000, C 0.000 }
gfCNCPoint6[2202] = {X 398.5577, Y 53.1200, Z -8.0000, A 0.000, B 0.000, C 0.000 }
gfCNCPoint6[2203] = {X 419.4886, Y 53.1200, Z -8.0000, A 0.000, B 0.000, C 0.000 }
gfCNCPoint6[2204] = {X 420.5533, Y 53.2376, Z -8.0000, A 0.000, B 0.000, C 0.000 }
gfCNCPoint6[2205] = {X 421.5666, Y 53.5846, Z -8.0000, A 0.000, B 0.000, C 0.000 }
gfCNCPoint6[2206] = {X 422.4799, Y 54.1443, Z -8.0000, A 0.000, B 0.000, C 0.000 }
gfCNCPoint6[2207] = {X 423.2490, Y 54.8898, Z -8.0000, A 0.000, B 0.000, C 0.000 }
gfCNCPoint6[2208] = {X 423.8370, Y 55.7851, Z -8.0000, A 0.000, B 0.000, C 0.000 }
gfCNCPoint6[2209] = {X 424.2155, Y 56.7871, Z -8.0000, A 0.000, B 0.000, C 0.000 }
gfCNCPoint6[2210] = {X 424.3662, Y 57.8476, Z -8.0000, A 0.000, B 0.000, C 0.000 }
gfCNCPoint6[2211] = {X 429.8191, Y 59.9719, Z -8.0000, A 0.000, B 0.000, C 0.000 }
gfCNCPoint6[2212] = {X 457.2978, Y 70.8748, Z -8.0000, A 0.000, B 0.000, C 0.000 }
gfCNCPoint6[2213] = {X 457.2980, Y 63.6738, Z -8.0000, A 0.000, B 0.000, C 0.000 }
gfCNCPoint6[2214] = {X 456.2901, Y 63.3053, Z -8.0000, A 0.000, B 0.000, C 0.000 }
gfCNCPoint6[2215] = {X 455.3870, Y 62.7253, Z -8.0000, A 0.000, B 0.000, C 0.000 }
gfCNCPoint6[2216] = {X 454.6326, Y 61.9620, Z -8.0000, A 0.000, B 0.000, C 0.000 }
gfCNCPoint6[2217] = {X 454.0633, Y 61.0523, Z -8.0000, A 0.000, B 0.000, C 0.000 }
gfCNCPoint6[2218] = {X 453.7066, Y 60.0401, Z -8.0000, A 0.000, B 0.000, C 0.000 }
gfCNCPoint6[2219] = {X 453.5798, Y 58.9744, Z -8.0000, A 0.000, B 0.000, C 0.000 }
gfCNCPoint6[2220] = {X 453.5796, Y 58.0000, Z -8.0000, A 0.000, B 0.000, C 0.000 }
gfCNCPoint6[2221] = {X 453.6734, Y 57.0480, Z -8.0000, A 0.000, B 0.000, C 0.000 }
gfCNCPoint6[2222] = {X 453.9511, Y 56.1325, Z -8.0000, A 0.000, B 0.000, C 0.000 }
gfCNCPoint6[2223] = {X 454.4020, Y 55.2888, Z -8.0000, A 0.000, B 0.000, C 0.000 }
gfCNCPoint6[2224] = {X 455.0089, Y 54.5493, Z -8.0000, A 0.000, B 0.000, C 0.000 }
gfCNCPoint6[2225] = {X 455.7484, Y 53.9424, Z -8.0000, A 0.000, B 0.000, C 0.000 }
gfCNCPoint6[2226] = {X 456.5921, Y 53.4915, Z -8.0000, A 0.000, B 0.000, C 0.000 }
gfCNCPoint6[2227] = {X 457.5076, Y 53.2138, Z -8.0000, A 0.000, B 0.000, C 0.000 }
gfCNCPoint6[2228] = {X 458.4596, Y 53.1200, Z -8.0000, A 0.000, B 0.000, C 0.000 }
gfCNCPoint6[2229] = {X 475.0000, Y 53.1200, Z -8.0000, A 0.000, B 0.000, C 0.000 }
gfCNCPoint6[2230] = {X 475.9520, Y 53.2138, Z -8.0000, A 0.000, B 0.000, C 0.000 }
gfCNCPoint6[2231] = {X 476.8675, Y 53.4915, Z -8.0000, A 0.000, B 0.000, C 0.000 }
gfCNCPoint6[2232] = {X 477.7112, Y 53.9424, Z -8.0000, A 0.000, B 0.000, C 0.000 }
gfCNCPoint6[2233] = {X 478.4507, Y 54.5493, Z -8.0000, A 0.000, B 0.000, C 0.000 }
gfCNCPoint6[2234] = {X 479.0576, Y 55.2888, Z -8.0000, A 0.000, B 0.000, C 0.000 }
gfCNCPoint6[2235] = {X 479.5085, Y 56.1325, Z -8.0000, A 0.000, B 0.000, C 0.000 }
gfCNCPoint6[2236] = {X 479.7862, Y 57.0480, Z -8.0000, A 0.000, B 0.000, C 0.000 }
gfCNCPoint6[2237] = {X 479.8800, Y 58.0000, Z -8.0000, A 0.000, B 0.000, C 0.000 }
gfCNCPoint6[2238] = {X 479.8798, Y 58.9744, Z -8.0000, A 0.000, B 0.000, C 0.000 }
gfCNCPoint6[2239] = {X 479.7530, Y 60.0401, Z -8.0000, A 0.000, B 0.000, C 0.000 }
gfCNCPoint6[2240] = {X 479.3963, Y 61.0524, Z -8.0000, A 0.000, B 0.000, C 0.000 }
gfCNCPoint6[2241] = {X 478.8269, Y 61.9622, Z -8.0000, A 0.000, B 0.000, C 0.000 }
gfCNCPoint6[2242] = {X 478.0724, Y 62.7255, Z -8.0000, A 0.000, B 0.000, C 0.000 }
gfCNCPoint6[2243] = {X 477.1693, Y 63.3054, Z -8.0000, A 0.000, B 0.000, C 0.000 }
gfCNCPoint6[2244] = {X 476.1612, Y 63.6739, Z -8.0000, A 0.000, B 0.000, C 0.000 }
gfCNCPoint6[2245] = {X 476.1617, Y 92.3304, Z -8.0000, A 0.000, B 0.000, C 0.000 }
gfCNCPoint6[2246] = {X 476.3603, Y 92.3885, Z -8.0000, A 0.000, B 0.000, C 0.000 }
gfCNCPoint6[2247] = {X 476.5574, Y 92.4515, Z -8.0000, A 0.000, B 0.000, C 0.000 }
gfCNCPoint6[2248] = {X 477.4770, Y 92.8685, Z -8.0000, A 0.000, B 0.000, C 0.000 }
gfCNCPoint6[2249] = {X 478.2905, Y 93.4665, Z -8.0000, A 0.000, B 0.000, C 0.000 }
gfCNCPoint6[2250] = {X 478.9628, Y 94.2197, Z -8.0000, A 0.000, B 0.000, C 0.000 }
gfCNCPoint6[2251] = {X 479.4649, Y 95.0957, Z -8.0000, A 0.000, B 0.000, C 0.000 }
gfCNCPoint6[2252] = {X 479.7751, Y 96.0565, Z -8.0000, A 0.000, B 0.000, C 0.000 }
gfCNCPoint6[2253] = {X 479.8800, Y 97.0606, Z -8.0000, A 0.000, B 0.000, C 0.000 }
gfCNCPoint6[2254] = {X 479.8800, Y 97.6952, Z -8.0000, A 0.000, B 0.000, C 0.000 }
gfCNCPoint6[2255] = {X 479.4000, Y 97.6952, Z -8.0000, A 0.000, B 0.000, C 0.000 }
gfCNCPoint6[2256] = {X 479.4000, Y 98.0000, Z -8.0000, A 0.000, B 0.000, C 0.000 }
gfCNCPoint6[2257] = {X 479.2897, Y 98.9791, Z -8.0000, A 0.000, B 0.000, C 0.000 }
gfCNCPoint6[2258] = {X 478.9643, Y 99.9091, Z -8.0000, A 0.000, B 0.000, C 0.000 }
gfCNCPoint6[2259] = {X 478.4401, Y 100.7434, Z -8.0000, A 0.000, B 0.000, C 0.000 }
gfCNCPoint6[2260] = {X 477.7434, Y 101.4401, Z -8.0000, A 0.000, B 0.000, C 0.000 }
gfCNCPoint6[2261] = {X 476.9091, Y 101.9643, Z -8.0000, A 0.000, B 0.000, C 0.000 }
gfCNCPoint6[2262] = {X 475.9791, Y 102.2897, Z -8.0000, A 0.000, B 0.000, C 0.000 }
gfCNCPoint6[2263] = {X 475.0000, Y 102.4000, Z -8.0000, A 0.000, B 0.000, C 0.000 }
gfCNCPoint6[2264] = {X 458.4596, Y 102.4000, Z -8.0000, A 0.000, B 0.000, C 0.000 }
gfCNCPoint6[2265] = {X 457.4805, Y 102.2897, Z -8.0000, A 0.000, B 0.000, C 0.000 }
gfCNCPoint6[2266] = {X 456.5505, Y 101.9643, Z -8.0000, A 0.000, B 0.000, C 0.000 }
gfCNCPoint6[2267] = {X 455.7162, Y 101.4401, Z -8.0000, A 0.000, B 0.000, C 0.000 }
gfCNCPoint6[2268] = {X 455.0195, Y 100.7434, Z -8.0000, A 0.000, B 0.000, C 0.000 }
gfCNCPoint6[2269] = {X 454.4953, Y 99.9091, Z -8.0000, A 0.000, B 0.000, C 0.000 }
gfCNCPoint6[2270] = {X 454.1699, Y 98.9791, Z -8.0000, A 0.000, B 0.000, C 0.000 }
gfCNCPoint6[2271] = {X 454.0596, Y 98.0000, Z -8.0000, A 0.000, B 0.000, C 0.000 }
gfCNCPoint6[2272] = {X 454.0596, Y 97.0659, Z -8.0000, A 0.000, B 0.000, C 0.000 }
gfCNCPoint6[2273] = {X 454.1492, Y 96.1826, Z -8.0000, A 0.000, B 0.000, C 0.000 }
gfCNCPoint6[2274] = {X 454.4143, Y 95.3353, Z -8.0000, A 0.000, B 0.000, C 0.000 }
gfCNCPoint6[2275] = {X 454.8440, Y 94.5584, Z -8.0000, A 0.000, B 0.000, C 0.000 }
gfCNCPoint6[2276] = {X 455.4210, Y 93.8836, Z -8.0000, A 0.000, B 0.000, C 0.000 }
gfCNCPoint6[2277] = {X 456.1217, Y 93.3384, Z -8.0000, A 0.000, B 0.000, C 0.000 }
gfCNCPoint6[2278] = {X 456.9176, Y 92.9450, Z -8.0000, A 0.000, B 0.000, C 0.000 }
gfCNCPoint6[2279] = {X 457.7763, Y 92.7193, Z -8.0000, A 0.000, B 0.000, C 0.000 }
gfCNCPoint6[2280] = {X 457.7763, Y 85.6495, Z -8.0000, A 0.000, B 0.000, C 0.000 }
gfCNCPoint6[2281] = {X 444.8695, Y 80.5900, Z -8.0000, A 0.000, B 0.000, C 0.000 }
gfCNCPoint6[2282] = {X 420.1046, Y 96.6319, Z -8.0000, A 0.000, B 0.000, C 0.000 }
gfCNCPoint6[2283] = {X 420.1067, Y 97.0659, Z -8.0000, A 0.000, B 0.000, C 0.000 }
gfCNCPoint6[2284] = {X 420.1067, Y 98.0000, Z -8.0000, A 0.000, B 0.000, C 0.000 }
gfCNCPoint6[2285] = {X 419.9964, Y 98.9791, Z -8.0000, A 0.000, B 0.000, C 0.000 }
gfCNCPoint6[2286] = {X 419.6710, Y 99.9091, Z -8.0000, A 0.000, B 0.000, C 0.000 }
gfCNCPoint6[2287] = {X 419.1468, Y 100.7434, Z -8.0000, A 0.000, B 0.000, C 0.000 }
gfCNCPoint6[2288] = {X 418.4501, Y 101.4401, Z -8.0000, A 0.000, B 0.000, C 0.000 }
gfCNCPoint6[2289] = {X 417.6158, Y 101.9643, Z -8.0000, A 0.000, B 0.000, C 0.000 }
gfCNCPoint6[2290] = {X 416.6858, Y 102.2897, Z -8.0000, A 0.000, B 0.000, C 0.000 }
gfCNCPoint6[2291] = {X 415.7067, Y 102.4000, Z -8.0000, A 0.000, B 0.000, C 0.000 }
gfCNCPoint6[2292] = {X 396.4059, Y 102.4000, Z -8.0000, A 0.000, B 0.000, C 0.000 }
gfCNCPoint6[2293] = {X 395.4269, Y 102.2897, Z -8.0000, A 0.000, B 0.000, C 0.000 }
gfCNCPoint6[2294] = {X 394.4969, Y 101.9643, Z -8.0000, A 0.000, B 0.000, C 0.000 }
gfCNCPoint6[2295] = {X 393.6626, Y 101.4401, Z -8.0000, A 0.000, B 0.000, C 0.000 }
gfCNCPoint6[2296] = {X 392.9659, Y 100.7434, Z -8.0000, A 0.000, B 0.000, C 0.000 }
gfCNCPoint6[2297] = {X 392.4417, Y 99.9091, Z -8.0000, A 0.000, B 0.000, C 0.000 }
gfCNCPoint6[2298] = {X 392.1163, Y 98.9791, Z -8.0000, A 0.000, B 0.000, C 0.000 }
gfCNCPoint6[2299] = {X 392.0059, Y 98.0000, Z -8.0000, A 0.000, B 0.000, C 0.000 }
gfCNCPoint6[2300] = {X 392.0059, Y 97.0659, Z -8.0000, A 0.000, B 0.000, C 0.000 }
gfCNCPoint6[2301] = {X 392.1157, Y 96.0893, Z -8.0000, A 0.000, B 0.000, C 0.000 }
gfCNCPoint6[2302] = {X 392.4395, Y 95.1613, Z -8.0000, A 0.000, B 0.000, C 0.000 }
gfCNCPoint6[2303] = {X 392.9612, Y 94.3284, Z -8.0000, A 0.000, B 0.000, C 0.000 }
gfCNCPoint6[2304] = {X 393.6548, Y 93.6321, Z -8.0000, A 0.000, B 0.000, C 0.000 }
gfCNCPoint6[2305] = {X 394.4856, Y 93.1071, Z -8.0000, A 0.000, B 0.000, C 0.000 }
gfCNCPoint6[2306] = {X 395.4123, Y 92.7796, Z -8.0000, A 0.000, B 0.000, C 0.000 }
gfCNCPoint6[2307] = {X 396.3885, Y 92.6660, Z -8.0000, A 0.000, B 0.000, C 0.000 }
gfCNCPoint6[2308] = {X 397.3379, Y 92.6231, Z -8.0000, A 0.000, B 0.000, C 0.000 }
gfCNCPoint6[2309] = {X 398.2840, Y 92.5335, Z -8.0000, A 0.000, B 0.000, C 0.000 }
gfCNCPoint6[2310] = {X 398.9176, Y 92.3799, Z -8.0000, A 0.000, B 0.000, C 0.000 }
gfCNCPoint6[2311] = {X 399.5010, Y 92.0886, Z -8.0000, A 0.000, B 0.000, C 0.000 }
gfCNCPoint6[2312] = {X 404.0994, Y 89.1252, Z -8.0000, A 0.000, B 0.000, C 0.000 }
gfCNCPoint6[2313] = {X 427.8776, Y 73.9167, Z -8.0000, A 0.000, B 0.000, C 0.000 }
gfCNCPoint6[2314] = {X 403.7263, Y 64.4417, Z -8.0000, A 0.000, B 0.000, C 0.000 }
gfCNCPoint6[2315] = {X 402.0391, Y 63.8832, Z -8.0000, A 0.000, B 0.000, C 0.000 }
gfCNCPoint6[2316] = {X 400.3009, Y 63.5125, Z -8.0000, A 0.000, B 0.000, C 0.000 }
gfCNCPoint6[2317] = {X 398.5326, Y 63.3340, Z -8.0000, A 0.000, B 0.000, C 0.000 }
gfCNCPoint6[2318] = {X 397.5577, Y 63.2189, Z -8.0000, A 0.000, B 0.000, C 0.000 }
gfCNCPoint6[2319] = {X 396.6325, Y 62.8905, Z -8.0000, A 0.000, B 0.000, C 0.000 }
gfCNCPoint6[2320] = {X 395.8032, Y 62.3652, Z -8.0000, A 0.000, B 0.000, C 0.000 }
gfCNCPoint6[2321] = {X 395.1110, Y 61.6690, Z -8.0000, A 0.000, B 0.000, C 0.000 }
gfCNCPoint6[2322] = {X 394.5904, Y 60.8367, Z -8.0000, A 0.000, B 0.000, C 0.000 }
gfCNCPoint6[2323] = {X 394.2672, Y 59.9097, Z -8.0000, A 0.000, B 0.000, C 0.000 }
gfCNCPoint6[2324] = {X 394.1577, Y 58.9341, Z -8.0000, A 0.000, B 0.000, C 0.000 }
gfCNCPoint6[2325] = {X 394.1577, Y 58.0000, Z -8.0000, A 0.000, B 0.000, C 0.000 }
gfCNCPoint6[2326] = {X 394.2680, Y 57.0209, Z -8.0000, A 0.000, B 0.000, C 0.000 }
gfCNCPoint6[2327] = {X 394.5935, Y 56.0909, Z -8.0000, A 0.000, B 0.000, C 0.000 }
gfCNCPoint6[2328] = {X 395.1177, Y 55.2566, Z -8.0000, A 0.000, B 0.000, C 0.000 }
gfCNCPoint6[2329] = {X 395.8144, Y 54.5599, Z -8.0000, A 0.000, B 0.000, C 0.000 }
gfCNCPoint6[2330] = {X 396.6486, Y 54.0357, Z -8.0000, A 0.000, B 0.000, C 0.000 }
gfCNCPoint6[2331] = {X 397.5786, Y 53.7103, Z -8.0000, A 0.000, B 0.000, C 0.000 }
gfCNCPoint6[2332] = {X 398.5577, Y 53.6000, Z -8.0000, A 0.000, B 0.000, C 0.000 }
gfCNCPoint6[2333] = {X 419.4886, Y 53.6000, Z -8.0000, A 0.000, B 0.000, C 0.000 }
gfCNCPoint6[2334] = {X 420.4677, Y 53.7103, Z -8.0000, A 0.000, B 0.000, C 0.000 }
gfCNCPoint6[2335] = {X 421.3977, Y 54.0357, Z -8.0000, A 0.000, B 0.000, C 0.000 }
gfCNCPoint6[2336] = {X 422.2320, Y 54.5599, Z -8.0000, A 0.000, B 0.000, C 0.000 }
gfCNCPoint6[2337] = {X 422.9287, Y 55.2566, Z -8.0000, A 0.000, B 0.000, C 0.000 }
gfCNCPoint6[2338] = {X 423.4529, Y 56.0909, Z -8.0000, A 0.000, B 0.000, C 0.000 }
gfCNCPoint6[2339] = {X 423.7783, Y 57.0209, Z -8.0000, A 0.000, B 0.000, C 0.000 }
gfCNCPoint6[2340] = {X 423.8886, Y 58.0000, Z -8.0000, A 0.000, B 0.000, C 0.000 }
gfCNCPoint6[2341] = {X 423.8886, Y 58.1767, Z -8.0000, A 0.000, B 0.000, C 0.000 }
gfCNCPoint6[2342] = {X 429.6420, Y 60.4180, Z -8.0000, A 0.000, B 0.000, C 0.000 }
gfCNCPoint6[2343] = {X 457.7778, Y 71.5817, Z -8.0000, A 0.000, B 0.000, C 0.000 }
gfCNCPoint6[2344] = {X 457.7781, Y 63.2810, Z -8.0000, A 0.000, B 0.000, C 0.000 }
gfCNCPoint6[2345] = {X 456.9191, Y 63.0556, Z -8.0000, A 0.000, B 0.000, C 0.000 }
gfCNCPoint6[2346] = {X 456.1228, Y 62.6623, Z -8.0000, A 0.000, B 0.000, C 0.000 }
gfCNCPoint6[2347] = {X 455.4218, Y 62.1171, Z -8.0000, A 0.000, B 0.000, C 0.000 }
gfCNCPoint6[2348] = {X 454.8445, Y 61.4422, Z -8.0000, A 0.000, B 0.000, C 0.000 }
gfCNCPoint6[2349] = {X 454.4144, Y 60.6652, Z -8.0000, A 0.000, B 0.000, C 0.000 }
gfCNCPoint6[2350] = {X 454.1492, Y 59.8176, Z -8.0000, A 0.000, B 0.000, C 0.000 }
gfCNCPoint6[2351] = {X 454.0596, Y 58.9341, Z -8.0000, A 0.000, B 0.000, C 0.000 }
gfCNCPoint6[2352] = {X 454.0596, Y 58.0000, Z -8.0000, A 0.000, B 0.000, C 0.000 }
gfCNCPoint6[2353] = {X 454.1699, Y 57.0209, Z -8.0000, A 0.000, B 0.000, C 0.000 }
gfCNCPoint6[2354] = {X 454.4953, Y 56.0909, Z -8.0000, A 0.000, B 0.000, C 0.000 }
gfCNCPoint6[2355] = {X 455.0195, Y 55.2566, Z -8.0000, A 0.000, B 0.000, C 0.000 }
gfCNCPoint6[2356] = {X 455.7162, Y 54.5599, Z -8.0000, A 0.000, B 0.000, C 0.000 }
gfCNCPoint6[2357] = {X 456.5505, Y 54.0357, Z -8.0000, A 0.000, B 0.000, C 0.000 }
gfCNCPoint6[2358] = {X 457.4805, Y 53.7103, Z -8.0000, A 0.000, B 0.000, C 0.000 }
gfCNCPoint6[2359] = {X 458.4596, Y 53.6000, Z -8.0000, A 0.000, B 0.000, C 0.000 }
gfCNCPoint6[2360] = {X 475.0000, Y 53.6000, Z -8.0000, A 0.000, B 0.000, C 0.000 }
gfCNCPoint6[2361] = {X 475.9791, Y 53.7103, Z -8.0000, A 0.000, B 0.000, C 0.000 }
gfCNCPoint6[2362] = {X 476.9091, Y 54.0357, Z -8.0000, A 0.000, B 0.000, C 0.000 }
gfCNCPoint6[2363] = {X 477.7434, Y 54.5599, Z -8.0000, A 0.000, B 0.000, C 0.000 }
gfCNCPoint6[2364] = {X 478.4401, Y 55.2566, Z -8.0000, A 0.000, B 0.000, C 0.000 }
gfCNCPoint6[2365] = {X 478.9643, Y 56.0909, Z -8.0000, A 0.000, B 0.000, C 0.000 }
gfCNCPoint6[2366] = {X 479.2897, Y 57.0209, Z -8.0000, A 0.000, B 0.000, C 0.000 }
gfCNCPoint6[2367] = {X 479.4000, Y 58.0000, Z -8.0000, A 0.000, B 0.000, C 0.000 }
gfCNCPoint6[2368] = {X 479.3998, Y 58.9704, Z -8.0000, A 0.000, B 0.000, C 0.000 }
gfCNCPoint6[2369] = {X 479.3040, Y 59.8482, Z -8.0000, A 0.000, B 0.000, C 0.000 }
gfCNCPoint6[2370] = {X 479.0348, Y 60.6891, Z -8.0000, A 0.000, B 0.000, C 0.000 }
gfCNCPoint6[2371] = {X 478.6032, Y 61.4594, Z -8.0000, A 0.000, B 0.000, C 0.000 }
gfCNCPoint6[2372] = {X 478.0264, Y 62.1279, Z -8.0000, A 0.000, B 0.000, C 0.000 }
gfCNCPoint6[2373] = {X 477.3278, Y 62.6679, Z -8.0000, A 0.000, B 0.000, C 0.000 }
gfCNCPoint6[2374] = {X 476.5354, Y 63.0575, Z -8.0000, A 0.000, B 0.000, C 0.000 }
gfCNCPoint6[2375] = {X 475.6812, Y 63.2810, Z -8.0000, A 0.000, B 0.000, C 0.000 }
gfCNCPoint6[2376] = {X 475.6817, Y 92.7033, Z -8.0000, A 0.000, B 0.000, C 0.000 }
gfCNCPoint6[2377] = {X 476.0461, Y 92.7965, Z -8.0000, A 0.000, B 0.000, C 0.000 }
gfCNCPoint6[2378] = {X 476.4057, Y 92.9069, Z -8.0000, A 0.000, B 0.000, C 0.000 }
gfCNCPoint6[2379] = {X 477.2344, Y 93.2827, Z -8.0000, A 0.000, B 0.000, C 0.000 }
gfCNCPoint6[2380] = {X 477.9675, Y 93.8216, Z -8.0000, A 0.000, B 0.000, C 0.000 }
gfCNCPoint6[2381] = {X 478.5734, Y 94.5004, Z -8.0000, A 0.000, B 0.000, C 0.000 }
gfCNCPoint6[2382] = {X 479.0259, Y 95.2898, Z -8.0000, A 0.000, B 0.000, C 0.000 }
gfCNCPoint6[2383] = {X 479.3055, Y 96.1557, Z -8.0000, A 0.000, B 0.000, C 0.000 }
gfCNCPoint6[2384] = {X 479.4000, Y 97.0606, Z -8.0000, A 0.000, B 0.000, C 0.000 }
gfCNCPoint6[2385] = {X 479.4000, Y 97.6952, Z -8.0000, A 0.000, B 0.000, C 0.000 }
gfCNCPoint6[2386] = {X 479.8800, Y 97.6952, Z -8.0000, A 0.000, B 0.000, C 0.000 }
gfCNCPoint6[2387] = {X 507.6811, Y 97.6952, Z -8.0000, A 0.000, B 0.000, C 0.000 }
gfCNCPoint6[2388] = {X 507.6811, Y 100.0952, Z -8.0000, A 0.000, B 0.000, C 0.000 }
gfCNCPoint6[2389] = {X 600.0147, Y 100.0952, Z -8.0000, A 0.000, B 0.000, C 0.000 }
gfCNCPoint6[2390] = {X 600.0672, Y 100.0699, Z -8.0000, A 0.000, B 0.000, C 0.000 }
gfCNCPoint6[2391] = {X 600.0950, Y 100.0186, Z -8.0000, A 0.000, B 0.000, C 0.000 }
gfCNCPoint6[2392] = {X 600.0967, Y 99.1432, Z -8.0000, A 0.000, B 0.000, C 0.000 }
gfCNCPoint6[2393] = {X 600.0967, Y 49.8790, Z -8.0000, A 0.000, B 0.000, C 0.000 }
gfCNCPoint6[2394] = {X 601.1113, Y 49.7518, Z -8.0000, A 0.000, B 0.000, C 0.000 }
gfCNCPoint6[2395] = {X 602.0771, Y 49.4159, Z -8.0000, A 0.000, B 0.000, C 0.000 }
gfCNCPoint6[2396] = {X 602.9517, Y 48.8861, Z -8.0000, A 0.000, B 0.000, C 0.000 }
gfCNCPoint6[2397] = {X 603.6967, Y 48.1857, Z -8.0000, A 0.000, B 0.000, C 0.000 }
gfCNCPoint6[2398] = {X 603.6967, Y 47.3863, Z -8.0000, A 0.000, B 0.000, C 0.000 }
gfCNCPoint6[2399] = {X 603.1504, Y 48.0716, Z -8.0000, A 0.000, B 0.000, C 0.000 }
gfCNCPoint6[2400] = {X 602.4791, Y 48.6351, Z -8.0000, A 0.000, B 0.000, C 0.000 }
gfCNCPoint6[2401] = {X 601.7095, Y 49.0543, Z -8.0000, A 0.000, B 0.000, C 0.000 }
gfCNCPoint6[2402] = {X 600.8721, Y 49.3127, Z -8.0000, A 0.000, B 0.000, C 0.000 }
gfCNCPoint6[2403] = {X 600.0000, Y 49.4000, Z -8.0000, A 0.000, B 0.000, C 0.000 }
gfCNCPoint6[2404] = {X 593.5565, Y 49.4000, Z -8.0000, A 0.000, B 0.000, C 0.000 }
gfCNCPoint6[2405] = {X 592.5988, Y 49.2945, Z -8.0000, A 0.000, B 0.000, C 0.000 }
gfCNCPoint6[2406] = {X 591.6870, Y 48.9831, Z -8.0000, A 0.000, B 0.000, C 0.000 }
gfCNCPoint6[2407] = {X 590.8648, Y 48.4806, Z -8.0000, A 0.000, B 0.000, C 0.000 }
gfCNCPoint6[2408] = {X 590.1717, Y 47.8112, Z -8.0000, A 0.000, B 0.000, C 0.000 }
gfCNCPoint6[2409] = {X 589.6410, Y 47.0071, Z -8.0000, A 0.000, B 0.000, C 0.000 }
gfCNCPoint6[2410] = {X 589.3741, Y 46.3664, Z -8.0000, A 0.000, B 0.000, C 0.000 }
gfCNCPoint6[2411] = {X 589.2113, Y 45.6918, Z -8.0000, A 0.000, B 0.000, C 0.000 }
gfCNCPoint6[2412] = {X 589.1565, Y 45.0000, Z -8.0000, A 0.000, B 0.000, C 0.000 }
gfCNCPoint6[2413] = {X 589.1565, Y 44.0645, Z -8.0000, A 0.000, B 0.000, C 0.000 }
gfCNCPoint6[2414] = {X 589.2601, Y 43.1281, Z -8.0000, A 0.000, B 0.000, C 0.000 }
gfCNCPoint6[2415] = {X 589.5590, Y 42.2346, Z -8.0000, A 0.000, B 0.000, C 0.000 }
gfCNCPoint6[2416] = {X 590.0398, Y 41.4244, Z -8.0000, A 0.000, B 0.000, C 0.000 }
gfCNCPoint6[2417] = {X 590.6809, Y 40.7341, Z -8.0000, A 0.000, B 0.000, C 0.000 }
gfCNCPoint6[2418] = {X 590.6817, Y 33.9441, Z -8.0000, A 0.000, B 0.000, C 0.000 }
gfCNCPoint6[2419] = {X 585.5192, Y 46.6830, Z -8.0000, A 0.000, B 0.000, C 0.000 }
gfCNCPoint6[2420] = {X 585.4476, Y 46.8466, Z -8.0000, A 0.000, B 0.000, C 0.000 }
gfCNCPoint6[2421] = {X 585.3694, Y 47.0071, Z -8.0000, A 0.000, B 0.000, C 0.000 }
gfCNCPoint6[2422] = {X 584.8417, Y 47.8075, Z -8.0000, A 0.000, B 0.000, C 0.000 }
gfCNCPoint6[2423] = {X 584.1532, Y 48.4747, Z -8.0000, A 0.000, B 0.000, C 0.000 }
gfCNCPoint6[2424] = {X 583.3365, Y 48.9769, Z -8.0000, A 0.000, B 0.000, C 0.000 }
gfCNCPoint6[2425] = {X 582.4111, Y 49.2946, Z -8.0000, A 0.000, B 0.000, C 0.000 }
gfCNCPoint6[2426] = {X 581.4384, Y 49.4000, Z -8.0000, A 0.000, B 0.000, C 0.000 }
gfCNCPoint6[2427] = {X 580.4664, Y 49.2878, Z -8.0000, A 0.000, B 0.000, C 0.000 }
gfCNCPoint6[2428] = {X 579.5433, Y 48.9635, Z -8.0000, A 0.000, B 0.000, C 0.000 }
gfCNCPoint6[2429] = {X 578.7146, Y 48.4433, Z -8.0000, A 0.000, B 0.000, C 0.000 }
